// TIA Portal project "Plantilla_V18" (V18)

(* hardware
DEVICE "S71500/ET200MP station_1"  S7-1500 station
   slot 0: "Perfil soporte_0"  Rack  6ES7 590-1***0-0AA0
   slot 1: "PLC_1"  CPU 1516-3 PN/DP  6ES7 516-3AN01-0AB0  V2.1
      slot 3: "Display de la CPU_1"  6ES7591-1BA00-0AA0
   slot 2: "DI 32x24VDC HF_1"  DI 32x24VDC HF  6ES7 521-1BL00-0AB0  V2.1
   slot 3: "DQ 32x24VDC/0.5A HF_1"  DQ 32x24VDC/0.5A HF  6ES7 522-1BL01-0AB0  V1.0
   slot 4: "AI 8xU/I/RTD/TC ST_1"  AI 8xU/I/RTD/TC ST  6ES7 531-7KF00-0AB0  V2.1
   slot 5: "AQ 4xU/I ST_1"  AQ 4xU/I ST  6ES7 532-5HD00-0AB0  V2.1
*)

// ===== PLC "PLC_1"  CPU 1516-3 PN/DP =====

VAR_GLOBAL   // PLC tag table "Temporizadores y contadores"
   "Temp_barnizado" AT %T0 : Timer;
   "Temp_secado1_normal" AT %T1 : Timer;
   "Temp_pickandplace_s1" AT %T2 : Timer;
   "Temp_grabado_normal_p" AT %T4 : Timer;
   "Temp_grabado_lim_p" AT %T5 : Timer;
   "Temp_grabado_pickandplace" AT %T6 : Timer;
   "Temp_secado1_lim" AT %T7 : Timer;
   "Temp_secado1_pickandplace" AT %T8 : Timer;
   "Temp_plataforma_s1" AT %T9 : Timer;
   "Temp_plataforma_lectura_s1" AT %T10 : Timer;
   "Temp_pintado_lim" AT %T11 : Timer;
   "Temp_cinta" AT %T12 : Timer;
   "Contador_lecturas_defectuosas" AT %Z0 : Counter;
   "Temp_fugaz_21" AT %T13 : Timer;
   "Temp_plataforma_p" AT %T14 : Timer;
   "Temp_plataforma_b" AT %T15 : Timer;
   "Temp_plataforma_lectura_p" AT %T16 : Timer;
   "Temp_plataforma_lectura_b" AT %T17 : Timer;
   "Temp_pickandplace_p" AT %T18 : Timer;
   "Temp_pickandplace_b" AT %T19 : Timer;
   "Temp_grabado_lim_b" AT %T20 : Timer;
   "Temp_grabado_normal_b" AT %T21 : Timer;
   "Temp_grabado_normal_s1" AT %T22 : Timer;
   "Temp_grabado_lim_s1" AT %T23 : Timer;
END_VAR

VAR_GLOBAL   // PLC tag table "Entradas"
   "ON" AT %E0.0 : Bool;
   "EMER" AT %E0.2 : Bool;
   "rearme" AT %E0.3 : Bool;
   "START" AT %E0.4 : Bool;
   "Tablero_ajedrez" AT %E1.2 : Bool;
   "Pieza_cogida_robpp_s1" AT %E6.4 : Bool;
   "fin_secado1" AT %E3.6 : Bool;
   "fin_grabado_p" AT %E3.7 : Bool;
   "fin_grabado_b" AT %E4.0 : Bool;
   "fin_grabado_s1" AT %E4.1 : Bool;
   "fin_pintado" AT %E4.2 : Bool;
   "Home_robpp_s1" AT %E4.3 : Bool;
   "Home_robpp_gs1" AT %E4.4 : Bool;
   "Home_robpp_gp" AT %E4.5 : Bool;
   "Home_robpp_gb" AT %E4.6 : Bool;
   "Home_robpp_p" AT %E4.7 : Bool;
   "lectura_correcta_s1" AT %E5.0 : Bool;
   "lectura_incorrecta_s1" AT %E5.1 : Bool;
   "entra_s1" AT %E5.2 : Bool;
   "sigue_s1" AT %E5.3 : Bool;
   "vel_cinta_muestreada_bits" AT %EW4 : Int;
   "lectura_correcta_p" AT %E5.4 : Bool;
   "lectura_incorrecta_p" AT %E6.1 : Bool;
   "lectura_correcta_b" AT %E6.2 : Bool;
   "lectura_incorrecta_b" AT %E6.3 : Bool;
   "entra_p" AT %E6.5 : Bool;
   "sigue_p" AT %E6.7 : Bool;
   "entra_b" AT %E7.0 : Bool;
   "sigue_b" AT %E7.1 : Bool;
   "Pieza_cogida_robpp_gp" AT %E7.2 : Bool;
   "Pieza_cogida_robpp_gb" AT %E7.3 : Bool;
END_VAR

VAR_GLOBAL   // PLC tag table "Salidas"
   "Barnizar" AT %A0.0 : Bool;
   "Pintar" AT %A0.1 : Bool;
   "Secar" AT %A0.2 : Bool;
   "Robot_coger" AT %A0.3 : Bool;
   "Robot_dejar" AT %A0.4 : Bool;
   "Robot_reposo" AT %A0.5 : Bool;
   "Grabar" AT %A0.6 : Bool;
   "aviso_error_barnizado" AT %A0.7 : Bool;
   "aviso_fin_barnizado" AT %A1.1 : Bool;
   "aviso_error_secado1" AT %A1.2 : Bool;
   "aviso_fin_secado1" AT %A1.3 : Bool;
   "aviso_fin_pintado" AT %A1.4 : Bool;
   "aviso_error_grabado_p" AT %A1.5 : Bool;
   "aviso_fin_grabado_p" AT %A1.6 : Bool;
   "Robot_izq" AT %A1.7 : Bool;
   "Robot_delante" AT %A2.0 : Bool;
   "Robot_dcha" AT %A2.1 : Bool;
   "aviso_fin_pickandplace" AT %A2.2 : Bool;
   "aviso_errorT_pickandplace" AT %A2.3 : Bool;
   "aviso_errorConf_pickandplace" AT %A2.4 : Bool;
   "aviso_al_pp_coger_pieza_grabado_p" AT %A2.5 : Bool;
   "aviso_al_pp_coger_pieza_secado1" AT %A2.6 : Bool;
   "Leer" AT %A2.7 : Bool;
   "giro_ruedas_por_defecto" AT %A3.0 : Bool;
   "giro_ruedas_izquierda" AT %A3.1 : Bool;
   "aviso_errorT_lectura_plataforma_s1" AT %A3.2 : Bool;
   "avisor_errorT_plataforma_s1" AT %A3.3 : Bool;
   "aviso_fin_entrada_s1" AT %A3.4 : Bool;
   "aviso_fin_noEntra_s1" AT %A3.5 : Bool;
   "aviso_error_lectura_plataforma" AT %A3.6 : Bool;
   "aviso_error_pintado" AT %A1.0 : Bool;
   "cinta_sentido_antihorario" AT %A3.7 : Bool;
   "aviso_error_cinta" AT %A4.0 : Bool;
   "aviso_fin_cinta" AT %A4.1 : Bool;
   "Luz_Roja" AT %A4.2 : Bool;
   "aviso_fin_entrada_p" AT %A4.3 : Bool;
   "aviso_fin_entrada_b" AT %A4.4 : Bool;
   "aviso_fin_noEntra_p" AT %A4.5 : Bool;
   "aviso_fin_noEntra_b" AT %A4.6 : Bool;
   "aviso_fin_grabado_b" AT %A4.7 : Bool;
   "aviso_error_grabado_b" AT %A5.0 : Bool;
   "aviso_al_pp_coger_pieza_grabado_b" AT %A5.1 : Bool;
   "aviso_fin_grabado_s1" AT %A5.2 : Bool;
   "aviso_error_grabado_s1" AT %A5.3 : Bool;
   "aviso_al_pp_coger_pieza_grabsecado1" AT %A5.4 : Bool;
END_VAR

VAR_GLOBAL   // PLC tag table "Memorias"
   "M_flanco" AT %M0.0 : Bool;
   "PON" AT %M0.1 : Bool;
   "X0" AT %M0.2 : Bool;
   "X_ON" AT %M0.3 : Bool;
   "X_OFF" AT %M0.4 : Bool;
   "XM1" AT %M0.5 : Bool;
   "X1" AT %M0.6 : Bool;
   "XM2" AT %M0.7 : Bool;
   "X2" AT %M1.0 : Bool;
   "XM3" AT %M1.1 : Bool;
   "X3" AT %M1.2 : Bool;
   "XM4.1" AT %M1.3 : Bool;
   "X4.1" AT %M1.4 : Bool;
   "XM5.1" AT %M1.5 : Bool;
   "X5.1" AT %M1.6 : Bool;
   "XM6.1" AT %M1.7 : Bool;
   "X6.1" AT %M2.0 : Bool;
   "OFF" AT %E0.1 : Bool;
   "X_EMER" AT %M2.1 : Bool;
   "X10" AT %M2.2 : Bool;
   "X_PintadoModoCuadricula" AT %M2.3 : Bool;
   "X_PintadoModoNormal" AT %M2.4 : Bool;
   "X20" AT %M2.5 : Bool;
   "X21" AT %M2.6 : Bool;
   "X22" AT %M2.7 : Bool;
   "lectura_defectuosa" AT %M3.0 : Bool;
   "evento_lecturas" AT %M3.1 : Bool;
   "X23" AT %M3.2 : Bool;
   "XM7" AT %M3.3 : Bool;
   "X7" AT %M3.4 : Bool;
   "XM4.2" AT %M3.5 : Bool;
   "X4.2" AT %M3.6 : Bool;
   "XM4.3" AT %M3.7 : Bool;
   "X4.3" AT %M4.0 : Bool;
   "XM5.2" AT %M4.1 : Bool;
   "X5.2" AT %M4.2 : Bool;
   "XM5.3" AT %M4.3 : Bool;
   "X5.3" AT %M4.4 : Bool;
   "XM5.4" AT %M4.5 : Bool;
   "X5.4" AT %M4.6 : Bool;
   "X6.2" AT %M4.7 : Bool;
   "XM6.2" AT %M5.0 : Bool;
   "X6.3" AT %M5.1 : Bool;
   "XM6.3" AT %M5.2 : Bool;
   "X5.5" AT %M5.3 : Bool;
   "X5.6" AT %M5.4 : Bool;
   "X5.7" AT %M5.5 : Bool;
   "X5.8" AT %M5.6 : Bool;
   "XM5.5" AT %M5.7 : Bool;
   "XM5.6" AT %M6.0 : Bool;
   "XM5.7" AT %M6.1 : Bool;
   "XM5.8" AT %M6.2 : Bool;
END_VAR

VAR_GLOBAL   // PLC tag table "Entradas_SP"
   "SP_pintado_LaminaEnMesa" AT %E0.5 : Bool;
   "SP_barnizado_in" AT %E0.6 : Bool;
   "SP_secado1" AT %E0.7 : Bool;
   "SP_barnizado_out" AT %E1.3 : Bool;
   "SP_lectura_p" AT %E2.1 : Bool;
   "SP_lectura_b" AT %E2.2 : Bool;
   "SP_lectura_s1" AT %E2.3 : Bool;
   "SP_pickandplace_p_in" AT %E2.4 : Bool;
   "SP_pickandplace_p_out" AT %E2.5 : Bool;
   "SP_pickandplace_gp_in" AT %E2.6 : Bool;
   "SP_pickandplace_gp_out" AT %E2.7 : Bool;
   "SP_grabado_p" AT %E3.0 : Bool;
   "SP_grabado_b" AT %E3.1 : Bool;
   "SP_pickandplace_s1_in" AT %E6.0 : Bool;
   "SP_pickandplace_s1_out" AT %E1.1 : Bool;
   "SP_pickandplace_gs1_in" AT %E1.5 : Bool;
   "SP_pickandplace_gs1_out" AT %E3.2 : Bool;
   "SP_grabado_s1" AT %E3.3 : Bool;
   "SP_pickandplace_gb_in" AT %E3.4 : Bool;
   "SP_pickandplace_gb_out" AT %E3.5 : Bool;
   "SP_pintado_PiezaEnMesa" AT %E1.4 : Bool;
   "SP_pintado_LaminaEnOrigen" AT %E6.6 : Bool;
END_VAR

DATA_BLOCK "Datos_produccion"   // DB1
{ S7_Optimized_Access := 'TRUE' }
VERSION : 0.1
   VAR
      t_lim_respuesta_lectura : S5Time := S5T#10s;
      t_lim_plat_omni : S5Time := S5T#60s;
      t_lim_barnizado : S5Time := S5T#10s;
      t_lim_secado : S5Time := S5T#60s;
      t_normal_secado : S5Time := S5T#10s;
      t_lim_pickandplace : S5Time := S5T#60s;
      t_lim_robotpintado : S5Time := S5T#10s;
      t_lim_grabado : S5Time := S5T#60s;
      t_normal_grabado : S5Time := S5T#15s;
      t_lim_cinta : S5Time := S5T#10s;
      max_malas_lecturas : Word := 30;
      t_fugaz_21 : S5Time := S5T#1s;
      t_lim_pintado : S5Time;
   END_VAR
BEGIN
END_DATA_BLOCK

DATA_BLOCK "Datos_ModoCuadricula"   // DB20
{ S7_Optimized_Access := 'TRUE' }
VERSION : 0.1
   VAR
      t_lim_pintado_ModoCuadricula : S5Time := S5T#600s;
   END_VAR
BEGIN
END_DATA_BLOCK

DATA_BLOCK "Datos_ModoNormal"   // DB21
{ S7_Optimized_Access := 'TRUE' }
VERSION : 0.1
   VAR
      t_lim_pintado_ModoNormal : S5Time := S5T#180s;
   END_VAR
BEGIN
END_DATA_BLOCK

// folder: Barnizado

DATA_BLOCK "maniobra_barnizado_DB"   // DB2
{ S7_Optimized_Access := 'TRUE' }
VERSION : 0.1
// stored: InstanceOfName maniobra_barnizado
"maniobra_barnizado"
BEGIN
END_DATA_BLOCK

// folder: Cinta

DATA_BLOCK "maniobra_cinta_DB"   // DB8
{ S7_Optimized_Access := 'TRUE' }
VERSION : 0.1
// stored: InstanceOfName maniobra_cinta
"maniobra_cinta"
BEGIN
END_DATA_BLOCK

// folder: Entrada_a_estacion

DATA_BLOCK "maniobra_plataforma_omnidireccional_DB"   // DB6
{ S7_Optimized_Access := 'TRUE' }
VERSION : 0.1
// stored: InstanceOfName maniobra_plataforma_omnidireccional
"maniobra_plataforma_omnidireccional"
BEGIN
END_DATA_BLOCK

DATA_BLOCK "man_plat_omni_DB_Entrada_Pintado"   // DB7
{ S7_Optimized_Access := 'TRUE' }
VERSION : 0.1
// stored: InstanceOfName maniobra_plataforma_omnidireccional
"maniobra_plataforma_omnidireccional"
BEGIN
END_DATA_BLOCK

DATA_BLOCK "man_plat_omni_DB_Entrada_Barnizado"   // DB10
{ S7_Optimized_Access := 'TRUE' }
VERSION : 0.1
// stored: InstanceOfName maniobra_plataforma_omnidireccional
"maniobra_plataforma_omnidireccional"
BEGIN
END_DATA_BLOCK

// folder: Grabado_y_secado

DATA_BLOCK "maniobra_secado_DB"   // DB4
{ S7_Optimized_Access := 'TRUE' }
VERSION : 0.1
// stored: InstanceOfName maniobra_grabado_secado
"maniobra_grabado_secado"
BEGIN
END_DATA_BLOCK

DATA_BLOCK "maniobra_grabado_DB"   // DB5
{ S7_Optimized_Access := 'TRUE' }
VERSION : 0.1
// stored: InstanceOfName maniobra_grabado_secado
"maniobra_grabado_secado"
BEGIN
END_DATA_BLOCK

DATA_BLOCK "man_grabado_b"   // DB14
{ S7_Optimized_Access := 'TRUE' }
VERSION : 0.1
// stored: InstanceOfName maniobra_grabado_secado
"maniobra_grabado_secado"
BEGIN
END_DATA_BLOCK

// folder: Pick_and_place

DATA_BLOCK "maniobra_pickandplace_DB"   // DB3
{ S7_Optimized_Access := 'TRUE' }
VERSION : 0.1
// stored: InstanceOfName maniobra_pickandplace
"maniobra_pickandplace"
BEGIN
END_DATA_BLOCK

DATA_BLOCK "man_pickandplace_gp1"   // DB11
{ S7_Optimized_Access := 'TRUE' }
VERSION : 0.1
// stored: InstanceOfName maniobra_pickandplace
"maniobra_pickandplace"
BEGIN
END_DATA_BLOCK

DATA_BLOCK "man_pickandplace_gp2"   // DB12
{ S7_Optimized_Access := 'TRUE' }
VERSION : 0.1
// stored: InstanceOfName maniobra_pickandplace
"maniobra_pickandplace"
BEGIN
END_DATA_BLOCK

DATA_BLOCK "man_pickandplace_gb1"   // DB13
{ S7_Optimized_Access := 'TRUE' }
VERSION : 0.1
// stored: InstanceOfName maniobra_pickandplace
"maniobra_pickandplace"
BEGIN
END_DATA_BLOCK

DATA_BLOCK "man_pickandplace_gb2"   // DB15
{ S7_Optimized_Access := 'TRUE' }
VERSION : 0.1
// stored: InstanceOfName maniobra_pickandplace
"maniobra_pickandplace"
BEGIN
END_DATA_BLOCK

DATA_BLOCK "man_pickandplace_s1_2"   // DB16
{ S7_Optimized_Access := 'TRUE' }
VERSION : 0.1
// stored: InstanceOfName maniobra_pickandplace
"maniobra_pickandplace"
BEGIN
END_DATA_BLOCK

DATA_BLOCK "man_pickandplace_gs1_1"   // DB17
{ S7_Optimized_Access := 'TRUE' }
VERSION : 0.1
// stored: InstanceOfName maniobra_pickandplace
"maniobra_pickandplace"
BEGIN
END_DATA_BLOCK

DATA_BLOCK "man_grabado_s1"   // DB18
{ S7_Optimized_Access := 'TRUE' }
VERSION : 0.1
// stored: InstanceOfName maniobra_grabado_secado
"maniobra_grabado_secado"
BEGIN
END_DATA_BLOCK

DATA_BLOCK "man_pickandplace_gs1_2"   // DB19
{ S7_Optimized_Access := 'TRUE' }
VERSION : 0.1
// stored: InstanceOfName maniobra_pickandplace
"maniobra_pickandplace"
BEGIN
END_DATA_BLOCK

// folder: Pintado

DATA_BLOCK "maniobra_pintado_DB_1"   // DB9
{ S7_Optimized_Access := 'TRUE' }
VERSION : 0.1
// stored: InstanceOfName maniobra_pintado
"maniobra_pintado"
BEGIN
END_DATA_BLOCK

// folder: (top level)

ORGANIZATION_BLOCK "Main"   // OB1, STL, ProgramCycle
TITLE = "Main Program Sweep (Cycle)"
{ S7_Optimized_Access := 'TRUE' }
VERSION : 0.1
   VAR_INPUT
      Initial_Call : Bool;   // Initial call of this OB
      Remanence : Bool;   // =True, if remanent data are available
   END_VAR
BEGIN

REGION Network 1: Llamada a los tests unitarios (comentado)
   //CALL  "test_barnizado"

   // CALL  "test_secado"
   //   CALL  "test_grabado"
   //     CALL  "test_pickandplace"
   //     CALL  "test_plataforma_omnidireccional"
   //      CALL  "test_cinta"
   //      CALL  "test_pintado"
   //      CALL  "Modos_pintado"

   //   CALL  "Emergencia"
END_REGION

REGION Network 2: Llamada a las FC
         CALL  "contador_fallos_lectura"
         ( max_malas_lecturas  := "Datos_produccion".max_malas_lecturas,
           debe_retirar_piezas := "evento_lecturas"
         );
         CALL  "gestion_fallos_lectura";
         CALL  "Emergencia";
         CALL  "Flancos";
         CALL  "Modos_pintado";
END_REGION

REGION Network 3: X0 -> XM
         A     "X0";
         A     "PON";
         AN    "OFF";
         S     "XM1";
         S     "XM2";
         S     "XM3";
         S     "XM4.1";
         S     "XM4.2";
         S     "XM4.3";
         S     "XM5.1";
         S     "XM6.1";
         S     "XM7";
         S     "X_ON";
         R     "X0";
END_REGION

REGION Network 4: X_ON -> X_OFF
         A     "X_ON";
         A     "OFF";
         S     "X_OFF";
         R     "X_ON";
END_REGION

REGION Network 5: X1, X2, X3, X4, X5, X6, X7, X_OFF -> X0
         A     "X1";
         A     "X2";
         A     "X3";
         A     "X4.1";
         S     "XM4.2";
         S     "XM4.3";
         A     "X5.1";
         A     "X6.1";
         A     "X7";
         A     "X_OFF";
         S     "X0";
         R     "X1";
         R     "X2";
         R     "X3";
         R     "X4.1";
         R     "X4.2";
         R     "X4.3";
         R     "X5.1";
         R     "X6.1";
         R     "X7";
         R     "X_OFF";
END_REGION

REGION Network 6: X1 -> XM1
         A     "X1";
         A     "SP_pintado_PiezaEnMesa";
         S     "XM1";
         R     "X1";
END_REGION

REGION Network 7: X2 -> XM2
         A     "X2";
         A     "SP_barnizado_in";
         S     "XM2";
         R     "X2";
END_REGION

REGION Network 8: X3 -> XM3
         A     "X3";
         A     "SP_secado1";
         S     "XM3";
         R     "XM3";
END_REGION

REGION Network 9: X4.1-> XM4.1
         A     "X4.1";
         A     "SP_grabado_p";
         S     "XM4.1";
         R     "X4.1";
END_REGION

REGION Network 10: X4.2 -> XM4.2
         A     "X4.2";
         A     "SP_grabado_b";
         S     "XM4.2";
         R     "X4.2";
END_REGION

REGION Network 11: X4.3 -> XM4.3
         A     "X4.3";
         A     "SP_grabado_s1";
         S     "XM4.3";
         R     "X4.3";
END_REGION

REGION Network 12: X5.1-> XM5.1
         A     "X5.1";
         A     "SP_pickandplace_gb_in";
         S     "XM5.1";
         R     "X5.1";
END_REGION

REGION Network 13: X5.2->XM5.2
         A     "X5.2";
         A     "SP_pickandplace_gp_in";
         S     "XM5.2";
         R     "X5.2";
END_REGION

REGION Network 14: X5.3->XM5.3
         A     "X5.3";
         A     "SP_pickandplace_gb_in";
         R     "X5.3";
         S     "XM5.3";
END_REGION

REGION Network 15: X5.4->XM5.4
         A     "X5.4";
         A     "aviso_al_pp_coger_pieza_grabado_b";
         S     "XM5.4";
         R     "X5.4";
END_REGION

REGION Network 16: X5.5->XM5.5
         A     "X5.5";
         A     "SP_pickandplace_s1_in";
         R     "X5.5";
         S     "XM5.5";
END_REGION

REGION Network 17: X5.6->XM5.6
         A     "X5.6";
         A     "aviso_al_pp_coger_pieza_secado1";
         R     "X5.6";
         S     "XM5.6";
END_REGION

REGION Network 18: X5.7->XM5.7
         A     "X5.7";
         A     "SP_pickandplace_gs1_in";
         R     "X5.7";
         S     "XM5.7";
END_REGION

REGION Network 19: X5.8->XM5.8
         A     "X5.8";
         A     "aviso_al_pp_coger_pieza_grabsecado1";
         R     "X5.8";
         S     "XM5.8";
END_REGION

REGION Network 20: X6.1 -> XM6.1
         A     "X6.1";
         A     "X_ON";
         S     "XM6.1";
         R     "X6.1";
END_REGION

REGION Network 21: X6.2 -> XM6.2
         A     "X6.2";
         A     "X_ON";
         R     "X6.2";
         S     "XM6.2";
END_REGION

REGION Network 22: X6.3 -> XM6.3
         A     "X6.3";
         A     "X_ON";
         R     "X6.3";
         S     "XM6.3";
END_REGION

REGION Network 23: X7 -> XM7
         A     "X7";
         A     "X_ON";
         R     "X7";
         S     "XM7";
END_REGION

REGION Network 24: XM1 -> X1 y tratamiento M1 (pintado)
         A     "XM1";
         JCN   _pintado;
         CALL  "maniobra_pintado", "maniobra_pintado_DB_1"
         ( SP_pieza              := "SP_pintado_PiezaEnMesa",
           SP_lamina_mesa        := "SP_pintado_LaminaEnMesa",
           SP_lamina_pos_inicial := "SP_pintado_LaminaEnOrigen",
           ModoLamina            := "X_PintadoModoCuadricula",
           ModoNormal            := "X_PintadoModoNormal",
           pintado_terminado     := "fin_pintado",
           RESET                 := false,
           t_lim_pintado_con_lam := "Datos_produccion".t_lim_pintado_ModoCuadricula,
           t_lim_pintado_sin_lam := "Datos_produccion".t_lim_pintado_ModoNormal,
           Temporizador_limite   := "Temp_pintado_lim",
           Tempor_pickandplace1  := "Temp_pickandplace_s1",
           Tempor_pickandplace2  := "Temp_pickandplace_s1",
           SP_pickandplace_in    := "SP_pickandplace_p_in",
           SP_pickandplace_out   := "SP_pickandplace_p_out",
           Sensor_home           := "Home_robpp_p",
           Lamina_cogida         := "Pieza_cogida_robpp_s1",
           t_lim_pickandplace    := "Datos_produccion".t_lim_pickandplace,
           Act_pintar            := "Pintar",
           bde_tiempo            := "aviso_error_pintado",
           bdf_correcta          := "aviso_fin_pintado"
         );

         A     "aviso_fin_pintado";
         S     "X1";
         R     "XM1";
   _pintado:NOP   0;
END_REGION

REGION Network 25: XM2 -> X2 y tratamiento M2 (barnizado)
         A     "XM2";
         JCN   _barnizado;
         CALL  "maniobra_barnizado", "maniobra_barnizado_DB"
         ( SP               := "SP_barnizado_in",
           indicador_de_fin := "SP_barnizado_out",
           t_lim            := "Datos_produccion".t_lim_barnizado,
           Temporizador     := "Temp_barnizado",
           RESET            := false,
           Actuador         := "Barnizar",
           bde_tiempo       := "aviso_error_barnizado",
           bdf_correcta     := "aviso_fin_barnizado"
         );

         A     "aviso_fin_barnizado";
         S     "X2";
         R     "XM2";

   _barnizado:NOP   0;
END_REGION

REGION Network 26: XM3 -> X3 y tratamiento M3 (secado)
         A     "XM3";
         JCN   _secado;
         CALL  "maniobra_grabado_secado", "maniobra_secado_DB"
         ( SP_maq                   := "SP_secado1",
           t_normal_maq             := "Datos_produccion".t_normal_secado,
           t_lim_man                := "Datos_produccion".t_lim_secado,
           RESET                    := false,
           Temp_normal_maq          := "Temp_secado1_normal",
           Temp_lim_maq             := "Temp_secado1_lim",
           bdf_correcta             := "aviso_fin_secado1",
           bde_Tiempo               := "aviso_error_secado1",
           aviso_a_robot_para_coger := "aviso_al_pp_coger_pieza_secado1",
           Actuador                 := "Secar"
         );
         A     "aviso_fin_secado1";
         S     "X3";
         R     "XM3";
   _secado:NOP   0;
END_REGION

REGION Network 27: XM4.1 -> X4.1 y tratamiento M4.1 (grabado del pintado)
         A     "XM4.1";
         JCN   _grabadopintado;
         CALL  "maniobra_grabado_secado", "maniobra_grabado_DB"
         ( SP_maq                   := "SP_grabado_p",
           t_normal_maq             := "Datos_produccion".t_normal_grabado,
           t_lim_man                := "Datos_produccion".t_lim_grabado,
           RESET                    := FALSE,
           Temp_normal_maq          := "Temp_grabado_normal_p",
           Temp_lim_maq             := "Temp_grabado_lim_p",
           bdf_correcta             := "aviso_fin_grabado_p",
           bde_Tiempo               := "aviso_error_grabado_p",
           aviso_a_robot_para_coger := "aviso_al_pp_coger_pieza_grabado_p",
           Actuador                 := "Grabar"
         );
         A     "aviso_fin_grabado_p";
         S     "X4.1";
         R     "XM4.1";
   _grabadopintado:NOP   0;
END_REGION

REGION Network 28: XM4.2 -> X4.2 y tratamiento M4.2 (grabado del barnizado)
         A     "XM4.2";
         JCN   _grabadobarnizado;
         CALL  "maniobra_grabado_secado", "man_grabado_b"
         ( SP_maq                   := "SP_grabado_b",
           t_normal_maq             := "Datos_produccion".t_normal_grabado,
           t_lim_man                := "Datos_produccion".t_lim_grabado,
           RESET                    := false,
           Temp_normal_maq          := "Temp_grabado_normal_b",
           Temp_lim_maq             := "Temp_grabado_lim_b",
           bdf_correcta             := "aviso_fin_grabado_b",
           bde_Tiempo               := "aviso_error_grabado_b",
           aviso_a_robot_para_coger := "aviso_al_pp_coger_pieza_grabado_b",
           Actuador                 := "Grabar"
         );
         A     "aviso_fin_grabado_b";
         S     "X4.2";
         R     "XM4.2";
   _grabadobarnizado:NOP   0;
END_REGION

REGION Network 29: XM4.3 -> X4.3 y tratamiento M4.3 (grabado del secado)
         A     "XM4.3";
         JCN   _grabadosecado;
         CALL  "maniobra_grabado_secado", "man_grabado_s1"
         ( SP_maq                   := "SP_grabado_s1",
           t_normal_maq             := "Datos_produccion".t_normal_grabado,
           t_lim_man                := "Datos_produccion".t_lim_grabado,
           RESET                    := false,
           Temp_normal_maq          := "Temp_grabado_normal_s1",
           Temp_lim_maq             := "Temp_grabado_lim_s1",
           bdf_correcta             := "aviso_fin_grabado_s1",
           bde_Tiempo               := "aviso_error_grabado_s1",
           aviso_a_robot_para_coger := "aviso_al_pp_coger_pieza_grabsecado1",
           Actuador                 := "Grabar"
         );
         A     "aviso_fin_grabado_s1";
         S     "X4.3";
         R     "XM4.3";
   _grabadosecado:NOP   0;
END_REGION

REGION Network 30: XM5.1->X5.1 y tratamiento M5.1 (pick and place para dejar pieza en la grabadora pintado)
         A     "XM5.1";
         JCN   _pickandplace_grabadopintado1;
         CALL  "maniobra_pickandplace", "man_pickandplace_gp1"
         ( SP1          := "SP_pickandplace_gb_in",
           P_cogida     := "Pieza_cogida_robpp_gp",
           S_home       := "Home_robpp_gp",
           t_lim        := "Datos_produccion".t_lim_pickandplace,
           Temporizador := "Temp_pickandplace_p",
           RESET        := false,
           SP2          := "SP_grabado_p",
           Mov1         := "Robot_coger",
           Mov2         := "Robot_delante",
           Mov4         := "Robot_reposo",
           bdf_correcta := "aviso_fin_pickandplace",
           bde_tiempo   := "aviso_errorT_pickandplace",
           bde_config   := "aviso_errorConf_pickandplace",
           Mov0         := "Robot_izq",
           Mov3         := "Robot_dejar"
         );
         A     "aviso_fin_pickandplace";
         S     "X5.1";
         R     "XM5.1";
   _pickandplace_grabadopintado1:NOP   0;
END_REGION

REGION Network 31: XM5.2->X5.2 y tratamiento M5.2 (pick and place para recoger la pieza de la grabadora de pintado)
         A     "XM5.2";
         JCN   _pickandplace_grabadopintado2;
         CALL  "maniobra_pickandplace", "man_pickandplace_gp1"
         ( SP1          := "SP_pickandplace_gp_in",
           P_cogida     := "Pieza_cogida_robpp_gp",
           S_home       := "Home_robpp_gp",
           t_lim        := "Datos_produccion".t_lim_pickandplace,
           Temporizador := "Temp_pickandplace_p",
           RESET        := false,
           SP2          := "SP_grabado_p",
           Mov1         := "Robot_coger",
           Mov2         := "Robot_delante",
           Mov4         := "Robot_reposo",
           bdf_correcta := "aviso_fin_pickandplace",
           bde_tiempo   := "aviso_errorT_pickandplace",
           bde_config   := "aviso_errorConf_pickandplace",
           Mov0         := "Robot_izq",
           Mov3         := "Robot_dejar"
         );
         A     "aviso_fin_pickandplace";
         R     "XM5.2";
         S     "X5.2";
   _pickandplace_grabadopintado2:NOP   0;
END_REGION

REGION Network 32: XM5.3->X5.3 y tratamiento M5.3 (pick and place para meter la pieza en la grabadora de barnizado)
         A     "XM5.3";
         JCN   _pickandplace_grabado_barnizado1;
         CALL  "maniobra_pickandplace", "man_pickandplace_gb1"
         ( SP1          := "SP_pickandplace_gb_in",
           P_cogida     := "Pieza_cogida_robpp_gb",
           S_home       := "Home_robpp_gb",
           t_lim        := "Datos_produccion".t_lim_pickandplace,
           Temporizador := "Temp_pickandplace_b",
           RESET        := false,
           SP2          := "SP_grabado_b",
           Mov1         := "Robot_coger",
           Mov2         := "Robot_delante",
           Mov4         := "Robot_reposo",
           bdf_correcta := "aviso_fin_pickandplace",
           bde_tiempo   := "aviso_errorT_pickandplace",
           bde_config   := "aviso_errorConf_pickandplace",
           Mov0         := "Robot_izq",
           Mov3         := "Robot_dejar"
         );
         A     "aviso_fin_pickandplace";
         S     "X5.3";
         R     "XM5.3";
   _pickandplace_grabado_barnizado1:NOP   0;
END_REGION

REGION Network 33: XM5.4->X5.4 y tratamiento M5.4 (pick and place para recoger la pieza del grabado del barnizado)
         A     "XM5.4";
         JCN   _pickandplace_grabado_barnizado2;
         CALL  "maniobra_pickandplace", "man_pickandplace_gb2"
         ( SP1          := "aviso_al_pp_coger_pieza_grabado_b",
           P_cogida     := "Pieza_cogida_robpp_gb",
           S_home       := "Home_robpp_gb",
           t_lim        := "Datos_produccion".t_lim_pickandplace,
           Temporizador := "Temp_pickandplace_b",
           RESET        := false,
           SP2          := "SP_pickandplace_gb_out",
           Mov1         := "Robot_coger",
           Mov2         := "Robot_dcha",
           Mov4         := "Robot_reposo",
           bdf_correcta := "aviso_fin_pickandplace",
           bde_tiempo   := "aviso_errorT_pickandplace",
           bde_config   := "aviso_errorConf_pickandplace",
           Mov0         := "Robot_delante",
           Mov3         := "Robot_dejar"
         );
         A     "aviso_fin_pickandplace";
         S     "X5.4";
         R     "XM5.4";
   _pickandplace_grabado_barnizado2:NOP   0;
END_REGION

REGION Network 34: XM5.5->X5.5 y tratamiento M5.5 (pick and place para meter la pieza en la máquina de secado)
         A     "XM5.5";
         JCN   _pickandplace_secado1;
         CALL  "maniobra_pickandplace", "maniobra_pickandplace_DB"
         ( SP1          := "SP_pickandplace_s1_in",
           P_cogida     := "Pieza_cogida_robpp_s1",
           S_home       := "Home_robpp_s1",
           t_lim        := "Datos_produccion".t_lim_pickandplace,
           Temporizador := "Temp_pickandplace_s1",
           RESET        := FALSE,
           SP2          := "SP_secado1",
           Mov1         := "Robot_coger",
           Mov2         := "Robot_delante",
           Mov4         := "Robot_reposo",
           bdf_correcta := "aviso_fin_pickandplace",
           bde_tiempo   := "aviso_errorT_pickandplace",
           bde_config   := "aviso_errorConf_pickandplace",
           Mov0         := "Robot_izq",
           Mov3         := "Robot_dejar"
         );
         A     "aviso_fin_pickandplace";
         R     "XM5.5";
         S     "X5.5";
   _pickandplace_secado1:NOP   0;
END_REGION

REGION Network 35: XM5.6->X5.6 y tratamiento M5.6 (pick and place para sacar la pieza de la máquina de secado)
         A     "XM5.6";
         JCN   _pickandplace_secado2;
         CALL  "maniobra_pickandplace", "man_pickandplace_s1_2"
         ( SP1          := "aviso_al_pp_coger_pieza_secado1",
           P_cogida     := "Pieza_cogida_robpp_s1",
           S_home       := "Home_robpp_s1",
           t_lim        := "Datos_produccion".t_lim_pickandplace,
           Temporizador := "Temp_pickandplace_s1",
           RESET        := false,
           SP2          := "SP_pickandplace_s1_out",
           Mov1         := "Robot_coger",
           Mov2         := "Robot_dcha",
           Mov4         := "Robot_reposo",
           bdf_correcta := "aviso_fin_pickandplace",
           bde_tiempo   := "aviso_errorT_pickandplace",
           bde_config   := "aviso_errorConf_pickandplace",
           Mov0         := "Robot_delante",
           Mov3         := "Robot_dejar"
         );
         A     "aviso_fin_pickandplace";
         R     "XM5.6";
         S     "X5.6";
   _pickandplace_secado2:NOP   0;
END_REGION

REGION Network 36: XM5.7->X5.7 y tratamiento M5.7 (pick and place para meter la pieza en la grabadora de secado)
         A     "XM5.7";
         JCN   _pickandplace_grabado_secado1;
         CALL  "maniobra_pickandplace", "man_pickandplace_gs1_1"
         ( SP1          := "SP_pickandplace_gs1_in",
           P_cogida     := "Pieza_cogida_robpp_s1",
           S_home       := "Home_robpp_s1",
           t_lim        := "Datos_produccion".t_lim_pickandplace,
           Temporizador := "Temp_pickandplace_s1",
           RESET        := false,
           SP2          := "SP_grabado_s1",
           Mov1         := "Robot_coger",
           Mov2         := "Robot_delante",
           Mov4         := "Robot_reposo",
           bdf_correcta := "aviso_fin_pickandplace",
           bde_tiempo   := "aviso_errorT_pickandplace",
           bde_config   := "aviso_errorConf_pickandplace",
           Mov0         := "Robot_izq",
           Mov3         := "Robot_dejar"
         );
         A     "aviso_fin_pickandplace";
         R     "XM5.7";
         S     "X5.7";
   _pickandplace_grabado_secado1:NOP   0;
END_REGION

REGION Network 37: XM5.78->X5.8 y tratamiento M5.8 (pick and place para sacar la pieza de la grabadora de secado)
         A     "XM5.8";
         JCN   _pickandplace_grabado_secado2;
         CALL  "maniobra_pickandplace", "man_pickandplace_gs1_2"
         ( SP1          := "aviso_al_pp_coger_pieza_grabsecado1",
           P_cogida     := "Pieza_cogida_robpp_s1",
           S_home       := "Home_robpp_s1",
           t_lim        := "Datos_produccion".t_lim_pickandplace,
           Temporizador := "Temp_pickandplace_s1",
           RESET        := false,
           SP2          := "SP_pickandplace_gs1_out",
           Mov1         := "Robot_coger",
           Mov2         := "Robot_dcha",
           Mov4         := "Robot_reposo",
           bdf_correcta := "aviso_fin_pickandplace",
           bde_tiempo   := "aviso_errorT_pickandplace",
           bde_config   := "aviso_errorConf_pickandplace",
           Mov0         := "Robot_delante",
           Mov3         := "Robot_dejar"
         );
         A     "aviso_fin_pickandplace";
         S     "X5.8";
         R     "XM5.8";

   _pickandplace_grabado_secado2:NOP   0;
END_REGION

REGION Network 38: XM6.1 -> X6.1 y tratamiento M6.1 (entrada a estación de pintado)
         A     "XM6.1";
         JCN   _entrada_pintado;
         CALL  "maniobra_plataforma_omnidireccional", "man_plat_omni_DB_Entrada_Pintado"
         ( SP                          := "SP_lectura_p",
           Lectura_correcta            := "lectura_correcta_p",
           Lectura_incorrecta          := "lectura_incorrecta_p",
           Entra_estacion              := "entra_p",
           Sigue_cinta                 := "sigue_p",
           SP_estacion                 := "SP_pickandplace_p_in",
           RESET                       := false,
           t_lim_lectura               := "Datos_produccion".t_lim_respuesta_lectura,
           t_lim_maniobra              := "Datos_produccion".t_lim_plat_omni,
           Temp_lectura                := "Temp_plataforma_lectura_p",
           Temp_maniobra               := "Temp_plataforma_p",
           Actuador_ruedas_por_defecto := "giro_ruedas_por_defecto",
           Actuador_lectura            := "Leer",
           Actuador_ruedas_giro        := "giro_ruedas_izquierda",
           bde_tiempo_lectura          := "aviso_errorT_lectura_plataforma_s1",
           bde_tiempo                  := "aviso_errorT_lectura_plataforma_s1",
           bde_lectura                 := "aviso_error_lectura_plataforma",
           bdf_piezadentro             := "aviso_fin_entrada_p",
           bdf_piezasiguerecto         := "aviso_fin_noEntra_p"
         );

         A     "aviso_fin_entrada_p";
         O     "aviso_fin_entrada_p";
         R     "XM6.1";
         S     "X6.1";
   _entrada_pintado:NOP   0;
END_REGION

REGION Network 39: XM6.2 -> X6.2 y tratamiento M6.2 (entrada a estación de barnizado)
         A     "XM6.2";
         JCN   _entrada_barnizado;
         CALL  "maniobra_plataforma_omnidireccional", "man_plat_omni_DB_Entrada_Barnizado"
         ( SP                          := "SP_lectura_b",
           Lectura_correcta            := "lectura_correcta_b",
           Lectura_incorrecta          := "lectura_incorrecta_b",
           Entra_estacion              := "entra_b",
           Sigue_cinta                 := "sigue_b",
           SP_estacion                 := "SP_barnizado_in",
           RESET                       := false,
           t_lim_lectura               := "Datos_produccion".t_lim_respuesta_lectura,
           t_lim_maniobra              := "Datos_produccion".t_lim_plat_omni,
           Temp_lectura                := "Temp_plataforma_lectura_b",
           Temp_maniobra               := "Temp_plataforma_b",
           Actuador_ruedas_por_defecto := "giro_ruedas_por_defecto",
           Actuador_lectura            := "Leer",
           Actuador_ruedas_giro        := "giro_ruedas_izquierda",
           bde_tiempo_lectura          := "aviso_errorT_lectura_plataforma_s1",
           bde_tiempo                  := "aviso_errorT_lectura_plataforma_s1",
           bde_lectura                 := "aviso_error_lectura_plataforma",
           bdf_piezadentro             := "aviso_fin_entrada_b",
           bdf_piezasiguerecto         := "aviso_fin_noEntra_b"
         );
         A     "aviso_fin_entrada_b";
         O     "aviso_fin_noEntra_b";
         R     "XM6.2";
         S     "X6.2";
   _entrada_barnizado:NOP   0;
END_REGION

REGION Network 40: XM6.3 -> X6.3 y tratamiento M6.3 (entrada a estación de secado)
         A     "XM6.3";
         JCN   _entrada_secado;
         CALL  "maniobra_plataforma_omnidireccional", "maniobra_plataforma_omnidireccional_DB"
         ( SP                          := "SP_lectura_s1",
           Lectura_correcta            := "lectura_correcta_s1",
           Lectura_incorrecta          := "lectura_incorrecta_s1",
           Entra_estacion              := "entra_s1",
           Sigue_cinta                 := "sigue_s1",
           SP_estacion                 := "SP_pickandplace_s1_in",
           RESET                       := false,
           t_lim_lectura               := "Datos_produccion".t_lim_respuesta_lectura,
           t_lim_maniobra              := "Datos_produccion".t_lim_plat_omni,
           Temp_lectura                := "Temp_plataforma_lectura_s1",
           Temp_maniobra               := "Temp_plataforma_s1",
           Actuador_ruedas_por_defecto := "giro_ruedas_por_defecto",
           Actuador_lectura            := "Leer",
           Actuador_ruedas_giro        := "giro_ruedas_izquierda",
           bde_tiempo_lectura          := "aviso_errorT_lectura_plataforma_s1",
           bde_tiempo                  := "avisor_errorT_plataforma_s1",
           bde_lectura                 := "aviso_error_lectura_plataforma",
           bdf_piezadentro             := "aviso_fin_entrada_s1",
           bdf_piezasiguerecto         := "aviso_fin_noEntra_s1"
         );
         A     "aviso_fin_entrada_s1";
         O     "aviso_fin_noEntra_s1";
         R     "XM6.3";
         S     "X6.3";
   _entrada_secado:NOP   0;
END_REGION

REGION Network 41: XM7 -> X7 y tratamiento de M7 (cinta)
         A     "XM7";
         JCN   _cinta;
         CALL  "maniobra_cinta", "maniobra_cinta_DB"
         ( vel_cinta_bits      := "vel_cinta_muestreada_bits",
           t_lim               := "Datos_produccion".t_lim_cinta,
           Temporizador        := "Temp_cinta",
           RESET               := "EMER",
           Sentido_antihorario := "cinta_sentido_antihorario",
           bdf_correcta        := "aviso_fin_cinta",
           bde_velocidad       := "aviso_error_cinta"
         );
         A     "aviso_fin_cinta";
         R     "XM7";
         S     "X7";
   _cinta:NOP   0;
END_REGION
END_ORGANIZATION_BLOCK

ORGANIZATION_BLOCK "Startup"   // OB100, STL, Startup
TITLE = "Complete Restart"
{ S7_Optimized_Access := 'TRUE' }
VERSION : 0.1
   VAR_INPUT
      LostRetentive : Bool;   // True if retentive data are lost
      LostRTC : Bool;   // True if date and time are lost
   END_VAR
BEGIN

REGION Network 1
         SET;
         S     "X0";
         S     "X10";
         S     "X20";
         R     "X_PintadoModoCuadricula";
         R     "X_PintadoModoNormal";
         R     "X_EMER";
         R     "X21";
         R     "X22";
END_REGION
END_ORGANIZATION_BLOCK

// folder: Barnizado

FUNCTION_BLOCK "maniobra_barnizado"   // FB2, STL
{ S7_Optimized_Access := 'TRUE' }
VERSION : 0.1
// Para reciclar código, se utiliza una misma maniobra para las máquinas de barnizado, grabado y secado.
   VAR_INPUT
      SP : Bool;
      indicador_de_fin : Bool;
      t_lim : S5Time := S5T#0ms;
      Temporizador : Timer;
      RESET : Bool;
   END_VAR
   VAR_OUTPUT
      Actuador : Bool;
      bde_tiempo : Bool;
      bdf_correcta : Bool;
   END_VAR
   VAR
      bdt : Bool;
      XE2 : Bool;
      X1 : Bool;
      XS2 : Bool;
      X_Err_Tiempo : Bool;
   END_VAR
BEGIN

REGION Network 1: Desconexión por RESET
         A     #RESET;
   //resetar los bits
         R     #bdt;
         R     #bde_tiempo;
         R     #bdf_correcta;
   //resetar temporizador
         R     #Temporizador;
         FR    #Temporizador;
   //resetar actuadores
         R     #Actuador;
         BEC;
END_REGION

REGION Network 2: Desconexión por error síncrono (exceso de tiempo)
         A     #X_Err_Tiempo;
         S     #bde_tiempo;
   //R     #X_Err_Tiempo
         R     #bdt;
         R     #bdf_correcta;
         R     #Temporizador;
         FR    #Temporizador;
         R     #Actuador;
         BEC;
END_REGION

REGION Network 3: Desconexión por finalización correcta
         A     #XS2;
         S     #bdf_correcta;
         R     #XS2;
         R     #bdt;
         R     #bde_tiempo;
         R     #Temporizador;
         FR    #Temporizador;
         R     #Actuador;
         BEC;
END_REGION

REGION Network 4: Conexión/ arranque de la maniobra
         SET;
         FP    #bdt;
         R     #bde_tiempo;
   //  R     #bdf_correcta
         S     #XE2;
         R     #X1;
         R     #XS2;
         R     #X_Err_Tiempo;
END_REGION

REGION Network 5: E2 -> X1
         A     #XE2;
         A     #SP;
         S     #X1;
         R     #XE2;
END_REGION

REGION Network 6: Definir perro guardián
         A     #X1;
         L     #t_lim;
         SS    #Temporizador;
END_REGION

REGION Network 7: X1-> XS2
         A     #X1;
         A     #indicador_de_fin;
         S     #XS2;
         R     #X1;
END_REGION

REGION Network 8: Activación del perro guardián
         A     #Temporizador;
         =     #X_Err_Tiempo;
END_REGION

REGION Network 9: Tratamiento X1
         A     #X1;
         =     #Actuador;
END_REGION
END_FUNCTION_BLOCK

// folder: Cinta

FUNCTION_BLOCK "maniobra_cinta"   // FB5, STL
{ S7_Optimized_Access := 'TRUE' }
VERSION : 0.1
   VAR_INPUT
      vel_cinta_bits : Int;
      t_lim : S5Time;
      Temporizador : Timer;
      RESET : Bool;
   END_VAR
   VAR_OUTPUT
      Sentido_antihorario : Bool;
      bdf_correcta : Bool;
      bde_velocidad : Bool;
   END_VAR
   VAR
      E7 : Bool;
      X1 : Bool;
      X2 : Bool;
      X_Err_Cinta : Bool;
      S7 : Bool;
      bdt : Bool;
      fuera_rango : Bool;
   END_VAR
   VAR_TEMP
      ret_val_scale : Word;
      vel_cinta_rpm : Real;
   END_VAR
BEGIN

REGION Network 1: Desconexión por RESET
         A     #RESET;
         R     #bdt;
         R     #bde_velocidad;
         R     #bdf_correcta;
         R     #Temporizador;
         FR    #Temporizador;
         R     #Sentido_antihorario;
         R     #fuera_rango;
         BEC;
END_REGION

REGION Network 2: Desconexión por velocidad de la cinta fuera de los rangos de lectura permitidos por el sensor
         A     #X_Err_Cinta;
         S     #bde_velocidad;
   // R     #X_Err_Cinta
         R     #bdt;
         R     #bdf_correcta;
         R     #Temporizador;
         FR    #Temporizador;
         R     #Sentido_antihorario;
         R     #fuera_rango;
         BEC;
END_REGION

REGION Network 3: Desconexión por finalización correcta
   // Si se mide un valor de velocidad fuera del rango, pero se corrige antes de que acabe el tiempo límite, se 
   // considera que la maniobra finaliza correctamente.
         A     #S7;
         S     #bdf_correcta;
   //R     #S7

         R     #bdt;
         R     #bde_velocidad;
         R     #Temporizador;
         FR    #Temporizador;
         R     #Sentido_antihorario;
         R     #fuera_rango;
         BEC;
END_REGION

REGION Network 4: Activación
         SET;
         FP    #bdt;

         R     #bdf_correcta;
         R     #bde_velocidad;

         S     #X1;
         R     #X2;
         R     #X_Err_Cinta;
         R     #S7;
END_REGION

REGION Network 5
         O     #X1;
         O     #X2;

         CALL  SCALE
         ( IN      := #vel_cinta_bits,
           HI_LIM  := 10000.0,
           LO_LIM  := 0.0,
           BIPOLAR := false,
           RET_VAL := #ret_val_scale,
           OUT     := #vel_cinta_rpm
         );
         O     #X1;
         O     #X2;
         A(;
         L     #ret_val_scale;
         L     W#16#0008;
         );
         ==I;
         =     #fuera_rango;
END_REGION

REGION Network 6: X1 ->X2
         A     #X1;
         A     #fuera_rango;
         S     #X2;
         R     #X1;
END_REGION

REGION Network 7: Configuración del temporizador
         A     #X2;
         L     #t_lim;
         SD    #Temporizador;
END_REGION

REGION Network 8: X2-> X_Err_Cinta
         A     #X2;
         A     #Temporizador;
         S     #X_Err_Cinta;
         R     #X2;
END_REGION

REGION Network 9: X2 -> S7
         A     #X2;
         AN    #fuera_rango;
         S     #S7;
         R     #X2;
END_REGION

REGION Network 10: Tratamiento de X1
         A     #X1;
         S     #Sentido_antihorario;
END_REGION

REGION Network 11: Tratamiento de X_Err_Cinta
         A     #X_Err_Cinta;
         R     #Sentido_antihorario;
END_REGION
END_FUNCTION_BLOCK

// folder: Emergencia

FUNCTION "Emergencia" : Void   // FC3, STL
{ S7_Optimized_Access := 'TRUE' }
VERSION : 0.1
BEGIN

REGION Network 1: Tratamiento de X_EMER
   // Se llama a todas las macroetapas, forzando como TRUE el valor de RESET, para que cada macroetapa haga la gestión de la emergencia.
         A     "EMER";
         JCN   _TratamientoEmergencia;
         CALL  "maniobra_barnizado", "maniobra_barnizado_DB"
         ( SP               := ,
           indicador_de_fin := ,
           t_lim            := ,
           Temporizador     := "Temp_barnizado",
           RESET            := true,
           Actuador         := "Barnizar",
           bde_tiempo       := "aviso_error_barnizado",
           bdf_correcta     := "aviso_fin_barnizado"
         );

         CALL  "maniobra_cinta", "maniobra_cinta_DB"
         ( vel_cinta_bits      := ,
           t_lim               := ,
           Temporizador        := "Temp_cinta",
           RESET               := true,
           Sentido_antihorario := "cinta_sentido_antihorario",
           bdf_correcta        := "aviso_fin_cinta",
           bde_velocidad       := "aviso_error_cinta"
         );

         CALL  "maniobra_grabado_secado", "maniobra_grabado_DB"
         ( SP_maq                   := ,
           t_normal_maq             := ,
           t_lim_man                := ,
           RESET                    := true,
           Temp_normal_maq          := "Temp_grabado_normal",
           Temp_lim_maq             := "Temp_grabado_lim",
           bdf_correcta             := "aviso_fin_grabado_p",
           bde_Tiempo               := "aviso_error_grabado_p",
           aviso_a_robot_para_coger := "aviso_al_pp_coger_pieza_grabado_p",
           Actuador                 := "Grabar"
         );

         CALL  "maniobra_grabado_secado", "maniobra_secado_DB"
         ( SP_maq                   := ,
           t_normal_maq             := ,
           t_lim_man                := ,
           RESET                    := true,
           Temp_normal_maq          := "Temp_secado1_normal",
           Temp_lim_maq             := "Temp_secado1_lim",
           bdf_correcta             := "aviso_fin_secado1",
           bde_Tiempo               := "aviso_error_secado1",
           aviso_a_robot_para_coger := "aviso_al_pp_coger_pieza_secado1",
           Actuador                 := "Secar"
         );

         CALL  "maniobra_pickandplace", "maniobra_pickandplace_DB"
         ( SP1          := ,
           P_cogida     := ,
           S_home       := ,
           t_lim        := ,
           Temporizador := "Temp_pickandplace",
           RESET        := true,
           SP2          := ,
           Mov1         := "Robot_coger",
           Mov2         := "Robot_delante",
           Mov4         := "Robot_reposo",
           bdf_correcta := "aviso_fin_pickandplace",
           bde_tiempo   := "aviso_errorT_pickandplace",
           bde_config   := "aviso_errorConf_pickandplace",
           Mov0         := "Robot_izq",
           Mov3         := "Robot_dejar"
         );


         CALL  "maniobra_pintado", "maniobra_pintado_DB_1"
         ( SP_pieza              := ,
           SP_lamina_mesa        := ,
           SP_lamina_pos_inicial := ,
           ModoLamina            := ,
           ModoNormal            := ,
           pintado_terminado     := ,
           RESET                 := true,
           t_lim_pintado_con_lam := ,
           t_lim_pintado_sin_lam := ,
           Temporizador_limite   := "Temp_pintado_lim",
           Tempor_pickandplace1  := "Temp_pickandplace",
           Tempor_pickandplace2  := "Temp_pickandplace",
           SP_pickandplace_in    := ,
           SP_pickandplace_out   := ,
           Sensor_home           := ,
           Lamina_cogida         := ,
           t_lim_pickandplace    := ,
           Act_pintar            := "Pintar",
           bde_tiempo            := "aviso_error_pintado",
           bdf_correcta          := "aviso_fin_pintado"
         );

         CALL  "maniobra_plataforma_omnidireccional", "maniobra_plataforma_omnidireccional_DB"
         ( SP                          := ,
           Lectura_correcta            := ,
           Lectura_incorrecta          := ,
           Entra_estacion              := ,
           Sigue_cinta                 := ,
           SP_estacion                 := ,
           RESET                       := true,
           t_lim_lectura               := ,
           t_lim_maniobra              := ,
           Temp_lectura                := "Temp_lectura_s1_in",
           Temp_maniobra               := "Temp_plataforma_s1",
           Actuador_ruedas_por_defecto := "giro_ruedas_por_defecto",
           Actuador_lectura            := "Leer",
           Actuador_ruedas_giro        := "giro_ruedas_izquierda",
           bde_tiempo_lectura          := "aviso_errorT_lectura_plataforma_s1",
           bde_tiempo                  := "aviso_errorT_lectura_plataforma_s1",
           bde_lectura                 := "aviso_error_lectura_plataforma",
           bdf_piezadentro             := "aviso_fin_entrada_s1",
           bdf_piezasiguerecto         := "aviso_fin_noEntra_s1"
         );

   _TratamientoEmergencia:NOP   0;

         A     "EMER";
         S     "X_EMER";

         R     "X1";
         R     "X2";
         R     "X3";
         R     "X4";
         R     "X5";
         R     "X6";
         R     "X_ON";
         R     "X_OFF";
         R     "X20";
         R     "X21";
         R     "X22";
         R     "X0";
         R     "XM1";
         R     "XM2";
         R     "XM3";
         R     "XM4";
         R     "XM5";
         R     "XM6";
         R     "X10";
         R     "X_PintadoModoCuadricula";
         R     "X_PintadoModoNormal";

         BEC;
END_REGION

REGION Network 2: Rearme de la celda mediante el pulsador de rearme sin estar la seta activada.
         A     "X_EMER";
         A     "rearme";
         AN    "EMER";
         S     "X0";
         R     "X_EMER";
END_REGION
END_FUNCTION

// folder: Entrada_a_estacion

FUNCTION_BLOCK "maniobra_plataforma_omnidireccional"   // FB7, STL
{ S7_Optimized_Access := 'TRUE' }
VERSION : 0.1
   VAR_INPUT
      SP : Bool;
      Lectura_correcta : Bool;
      Lectura_incorrecta : Bool;
      Entra_estacion : Bool;
      Sigue_cinta : Bool;
      SP_estacion : Bool;
      RESET : Bool;
      t_lim_lectura : S5Time;
      t_lim_maniobra : S5Time;
      Temp_lectura : Timer;
      Temp_maniobra : Timer;
   END_VAR
   VAR_OUTPUT
      Actuador_ruedas_por_defecto : Bool;
      Actuador_lectura : Bool;
      Actuador_ruedas_giro : Bool;
      bde_tiempo_lectura : Bool;
      bde_tiempo : Bool;
      bde_lectura : Bool;
      bdf_piezadentro : Bool;
      bdf_piezasiguerecto : Bool;
   END_VAR
   VAR
      XE5 : Bool;
      X1 : Bool;
      X2 : Bool;
      X3 : Bool;
      X4 : Bool;
      X_Err_TLectura : Bool;
      X_Err_Lectura : Bool;
      "XS5.1" : Bool;
      "XS5.2" : Bool;
      X_Err_Tiempo : Bool;
      bdt : Bool;
   END_VAR
BEGIN

REGION Network 1: Desconexión por RESET
         A     #RESET;

         R     #bdt;
         R     #bde_tiempo_lectura;
         R     #bdf_piezadentro;
         R     #bdf_piezasiguerecto;
         R     #bde_lectura;
         R     #bde_tiempo;

         R     #Temp_maniobra;
         FR    #Temp_maniobra;

         R     #Actuador_lectura;
         R     #Actuador_ruedas_giro;
         BEC;
END_REGION

REGION Network 2: Desconexión por error síncrono
         A     #X_Err_Tiempo;
         S     #bde_tiempo;
   //R     #X_Err_Tiempo

         R     #bdt;
         R     #bde_tiempo_lectura;
         R     #bdf_piezadentro;
         R     #bdf_piezasiguerecto;
         R     #bde_lectura;

         R     #Temp_maniobra;
         FR    #Temp_maniobra;

         R     #Actuador_lectura;
         R     #Actuador_ruedas_giro;
         BEC;
END_REGION

REGION Network 3: Desconexión por error por mala lectura
         A     #X_Err_Lectura;
         S     #bde_lectura;
   // R     #X_Err_Lectura

         R     #bdt;
         R     #bde_tiempo_lectura;
         R     #bdf_piezadentro;
         R     #bdf_piezasiguerecto;
         R     #bde_tiempo;

         R     #Temp_maniobra;
         FR    #Temp_maniobra;

         R     #Actuador_lectura;
         R     #Actuador_ruedas_giro;
         BEC;
END_REGION

REGION Network 4: Desconexión por error síncrono de lectura
         A     #X_Err_TLectura;
         S     #bde_tiempo_lectura;
   // R     #X_Err_TLectura

         R     #bdt;
         R     #bde_lectura;
         R     #bdf_piezadentro;
         R     #bdf_piezasiguerecto;
         R     #bde_tiempo;

         R     #Temp_maniobra;
         FR    #Temp_maniobra;

         R     #Actuador_lectura;
         R     #Actuador_ruedas_giro;
         BEC;
END_REGION

REGION Network 5: Desconexión por finalización correcta (pieza entra a la estación)
         A     #"XS5.1";
         S     #bdf_piezadentro;
   // R     #"XS5.1"

         R     #bdt;
         R     #bde_tiempo_lectura;
         R     #bdf_piezasiguerecto;
         R     #bde_lectura;
         R     #bde_tiempo;

         R     #Temp_maniobra;
         FR    #Temp_maniobra;

         R     #Actuador_lectura;
         R     #Actuador_ruedas_giro;
         BEC;
END_REGION

REGION Network 6: Desconexión por finalización correcta (pieza NO entra a la estación y sigue recto)
         A     #"XS5.2";
         S     #bdf_piezasiguerecto;
   //R     #"XS5.2"

         R     #bdt;
         R     #bde_tiempo_lectura;
         R     #bdf_piezadentro;
         R     #bde_lectura;
         R     #bde_tiempo;

         R     #Temp_maniobra;
         FR    #Temp_maniobra;

         R     #Actuador_lectura;
         R     #Actuador_ruedas_giro;
         BEC;
END_REGION

REGION Network 7: Conexión
         SET;
         FP    #bdt;

         R     #bdf_piezadentro;
         R     #bde_lectura;
         R     #bde_tiempo_lectura;
         R     #bde_tiempo;
         R     #bdf_piezasiguerecto;

         S     #XE5;
         S     #Actuador_ruedas_por_defecto;
         R     #X1;
         R     #X2;
         R     #X3;
         R     #"XS5.1";
         R     #"XS5.2";
         R     #X_Err_Lectura;
         R     #X_Err_Tiempo;
END_REGION

REGION Network 8: E5 -> X1
         A     #XE5;
         A     #SP;
         S     #X1;
         R     #XE5;
END_REGION

REGION Network 9: Configuración del perro guardián
         A     #X1;

         L     #t_lim_maniobra;
         SS    #Temp_maniobra;

         L     #t_lim_lectura;
         SD    #Temp_lectura;
END_REGION

REGION Network 10: X1 -> X_Err_Lectura
         A     #X1;
         A     #Temp_lectura;
         S     #X_Err_TLectura;
         R     #X1;
END_REGION

REGION Network 11: X1 -> X2
         A     #X1;
         A     #Lectura_correcta;
         AN    #Temp_lectura;
         S     #X2;
         R     #X1;
END_REGION

REGION Network 12: X1->X4
         A     #X1;
         A     #Lectura_incorrecta;
         AN    #Temp_lectura;
         S     #X4;
         R     #X1;
END_REGION

REGION Network 13: X2 -> X3
         A     #X2;
         A     #Entra_estacion;
         S     #X3;
         R     #X2;
         R     #Actuador_ruedas_por_defecto;
END_REGION

REGION Network 14: X3 -> S5.1
         A     #X3;
         A     #SP_estacion;
         R     #X3;
         S     #Actuador_ruedas_por_defecto;
         S     #"XS5.1";
END_REGION

REGION Network 15: X2 -> S5.2
         A     #X2;
         A     #Sigue_cinta;
         S     #"XS5.2";
         R     #X2;
END_REGION

REGION Network 16: Activación del perro guardián
         A     #Temp_maniobra;
         =     #X_Err_Tiempo;
END_REGION

REGION Network 17: Tratamiento X1
         A     #X1;
         =     #Actuador_lectura;
END_REGION

REGION Network 18: Tratamiento X3
         A     #X3;
         =     #Actuador_ruedas_giro;
END_REGION

REGION Network 19: Tratamiento X4
         A     #X4;
         =     #X_Err_Lectura;
END_REGION
END_FUNCTION_BLOCK

// folder: Flancos

FUNCTION "Flancos" : Void   // FC2, STL
{ S7_Optimized_Access := 'TRUE' }
VERSION : 0.1
BEGIN

REGION Network 1
         A     "ON";
         FP    "M_flanco";
         =     "PON";
END_REGION
END_FUNCTION

// folder: Grabado_y_secado

FUNCTION_BLOCK "maniobra_grabado_secado"   // FB3, STL
{ S7_Optimized_Access := 'TRUE' }
VERSION : 0.1
   VAR_INPUT
      SP_maq : Bool;
      t_normal_maq : S5Time;
      t_lim_man : S5Time;
      RESET : Bool;
      Temp_normal_maq : Timer;
      Temp_lim_maq : Timer;
   END_VAR
   VAR_OUTPUT
      bdf_correcta : Bool;
      bde_Tiempo : Bool;
      aviso_a_robot_para_coger : Bool;
      Actuador : Bool;
   END_VAR
   VAR
      XE3 : Bool;
      X1 : Bool;
      X2 : Bool;
      XS3 : Bool;
      X_Err_Tiempo_Man : Bool;
      bdt : Bool;
   END_VAR
BEGIN

REGION Network 1: Desconexión por RESET
         A     #RESET;

         R     #bdt;
         R     #bde_Tiempo;
         R     #bdf_correcta;

         R     #Temp_lim_maq;
         R     #Temp_normal_maq;
         FR    #Temp_lim_maq;
         FR    #Temp_normal_maq;

         R     #Actuador;
         R     #aviso_a_robot_para_coger;
         BEC;
END_REGION

REGION Network 2: Desonexión por error síncrono (exceso de tiempo en la maniobra de grabado o secado)
         A     #X_Err_Tiempo_Man;
         S     #bde_Tiempo;
   // R     #X_Err_Tiempo_Man

         R     #bdt;
         R     #bdf_correcta;

         R     #Temp_lim_maq;
         R     #Temp_normal_maq;
         FR    #Temp_lim_maq;
         FR    #Temp_normal_maq;

         R     #Actuador;
         R     #aviso_a_robot_para_coger;
         BEC;
END_REGION

REGION Network 3: Desconexión por finalización correcta de maniobra
         A     #XS3;
         S     #bdf_correcta;
   //R     #XS3
         R     #bdt;
         R     #bde_Tiempo;

         R     #Temp_lim_maq;
         R     #Temp_normal_maq;
         FR    #Temp_lim_maq;
         FR    #Temp_normal_maq;

         R     #Actuador;
         R     #aviso_a_robot_para_coger;
         BEC;
END_REGION

REGION Network 4: Conexión
         SET;
         FP    #bdt;

         R     #bde_Tiempo;
         R     #bdf_correcta;

         S     #XE3;
         R     #X1;
         R     #X2;
         R     #XS3;
         R     #X_Err_Tiempo_Man;
END_REGION

REGION Network 5: E3 -> X1
         A     #XE3;
         A     #SP_maq;
         S     #X1;
         R     #XE3;
END_REGION

REGION Network 6
         A     #X1;
         L     #t_normal_maq;
         SD    #Temp_normal_maq;

         L     #t_lim_man;
         SS    #Temp_lim_maq;
END_REGION

REGION Network 7: X1 -> X2
         A     #X1;
         A     #Temp_normal_maq;
         S     #X2;
         R     #X1;
END_REGION

REGION Network 8: X2 -> S3
         A     #X2;
         AN    #SP_maq;
         S     #XS3;
         R     #X2;
END_REGION

REGION Network 9: Activación del perro guardián por exceso de tiempo
         A     #Temp_lim_maq;
         =     #X_Err_Tiempo_Man;
END_REGION

REGION Network 10: Tratamiento de X1
         A     #X1;
         =     #Actuador;
END_REGION

REGION Network 11: Tratamiento de X2
         A     #X2;
         =     #aviso_a_robot_para_coger;
END_REGION
END_FUNCTION_BLOCK

// folder: Pick_and_place

FUNCTION_BLOCK "maniobra_pickandplace"   // FB4, STL
{ S7_Optimized_Access := 'TRUE' }
VERSION : 0.1
   VAR_INPUT
      SP1 : Bool;
      P_cogida : Bool;
      S_home : Bool;
      t_lim : S5Time;
      Temporizador : Timer;
      RESET : Bool;
      SP2 : Bool;
   END_VAR
   VAR_OUTPUT
      Mov1 : Bool;
      Mov2 : Bool;
      Mov4 : Bool;
      bdf_correcta : Bool;
      bde_tiempo : Bool;
      bde_config : Bool;
      Mov0 : Bool;
      Mov3 : Bool;
   END_VAR
   VAR
      XE4 : Bool;
      X1 : Bool;
      X2 : Bool;
      X3 : Bool;
      X4 : Bool;
      XS4 : Bool;
      X_Err_Tiempo : Bool;
      X_Err_Config : Bool;
      bdt : Bool;
   END_VAR
BEGIN

REGION Network 1: Desconexión por RESET
         A     #RESET;
   //resetar los bits
         R     #bdt;
         R     #bde_tiempo;
         R     #bde_config;
         R     #bdf_correcta;
   //resetar temporizador
         R     #Temporizador;
         FR    #Temporizador;
   //resetar actuadores
         R     #Mov0;
         R     #Mov1;
         R     #Mov2;
         R     #Mov3;
         R     #Mov4;
         BEC;
END_REGION

REGION Network 2: Desconexión por error síncrono
         A     #X_Err_Tiempo;
         S     #bde_tiempo;
   //R     #X_Err_Tiempo
         R     #bdt;
         R     #bdf_correcta;
         R     #bde_config;
         R     #Temporizador;
         FR    #Temporizador;
         R     #Mov0;
         R     #Mov1;
         R     #Mov2;
         R     #Mov3;
         R     #Mov4;
         BEC;
END_REGION

REGION Network 3: Desconexión por error de configuración
         A     #X_Err_Config;
         S     #bde_config;
   // R     #X_Err_Config
         R     #bdt;
         R     #bde_tiempo;
         R     #bdf_correcta;
         R     #Temporizador;
         FR    #Temporizador;
         R     #Mov0;
         R     #Mov1;
         R     #Mov2;
         R     #Mov3;
         R     #Mov4;

         BEC;
END_REGION

REGION Network 4: Desconexión por finalización correcta
         A     #XS4;
         S     #bdf_correcta;
   //R     #XS4
         R     #bdt;
         R     #bde_tiempo;
         R     #bde_config;
         R     #Temporizador;
         FR    #Temporizador;
         R     #Mov0;
         R     #Mov1;
         R     #Mov2;
         R     #Mov3;
         R     #Mov4;
         BEC;
END_REGION

REGION Network 5: Conexión
         SET;
         FP    #bdt;
         R     #bdf_correcta;
         R     #bde_config;
         R     #bde_tiempo;

         S     #XE4;
         R     #X1;
         R     #X2;
         R     #X3;
         R     #X4;
         R     #XS4;
         R     #X_Err_Config;
         R     #X_Err_Tiempo;
END_REGION

REGION Network 6: E4 -> X1
         A     #XE4;
         A     #SP1;
         S     #X1;
         R     #XE4;
END_REGION

REGION Network 7: Configuración del perro guardián
         A     #X4;  //cambiar a otro estado al finalizar test Q SINO NO ME DABA TIEMPO
         L     #t_lim;
         SS    #Temporizador;
END_REGION

REGION Network 8: X1 -> X2
         A     #X1;
         A     #P_cogida;
         S     #X2;
         R     #X1;
END_REGION

REGION Network 9: X2 -> X_Err_Config
   // Error por mala configuración: se produce cuando no se detecta la pieza cogida, cuando previamente se detectaba y no ha sido depositada,
   // es decir, cuando se cae de las pinzas.
         A     #X2;
         AN    #P_cogida;
         S     #X_Err_Config;
         R     #X2;
END_REGION

REGION Network 10: X2 -> X3
         A     #X2;
         A     #SP2;
         S     #X3;
         R     #X2;
END_REGION

REGION Network 11: X3 -> X4
         A     #X3;
         AN    #P_cogida;
         S     #X4;
         R     #X3;
END_REGION

REGION Network 12: X4 -> S4
         A     #X4;
         A     #S_home;
         S     #XS4;
         R     #X4;
END_REGION

REGION Network 13: Activación de perro guardián
         A     #Temporizador;
         =     #X_Err_Tiempo;
END_REGION

REGION Network 14
         A     #XE4;
         =     #Mov0;
END_REGION

REGION Network 15: Tratamiento de X1
         A     #X1;
         =     #Mov1;
END_REGION

REGION Network 16: Tratamiento de X2
         A     #X2;
         =     #Mov2;
END_REGION

REGION Network 17: Tratamiento de X3
         A     #X3;
         =     #Mov3;
END_REGION

REGION Network 18: Tratamiento de X4
         A     #X4;
         =     #Mov4;
END_REGION
END_FUNCTION_BLOCK

// folder: Pintado

FUNCTION_BLOCK "maniobra_pintado"   // FB6, STL
{ S7_Optimized_Access := 'TRUE' }
VERSION : 0.1
   VAR_INPUT
      SP_pieza : Bool;
      SP_lamina_mesa : Bool;
      SP_lamina_pos_inicial : Bool;
      ModoLamina : Bool;
      ModoNormal : Bool;
      pintado_terminado : Bool;
      RESET : Bool;
      t_lim_pintado_con_lam : S5Time;
      t_lim_pintado_sin_lam : S5Time;
      Temporizador_limite : Timer;
      Tempor_pickandplace1 : Timer;
      Tempor_pickandplace2 : Timer;
      SP_pickandplace_in : Bool;
      SP_pickandplace_out : Bool;
      Sensor_home : Bool;
      Lamina_cogida : Bool;
      t_lim_pickandplace : S5Time;
   END_VAR
   VAR_OUTPUT
      Act_pintar : Bool;
      bde_tiempo : Bool;
      bdf_correcta : Bool;
   END_VAR
   VAR
      usar_lamina : "maniobra_pickandplace";
      guardar_lamina : "maniobra_pickandplace";
      XE1 : Bool;
      X1 : Bool;
      XM1 : Bool;
      XM2 : Bool;
      X2 : Bool;
      X3 : Bool;
      XS1 : Bool;
      X_Err_Tiempo : Bool;
      bdt : Bool;
      Robot_lam_izq : Bool;
      Robot_lam_coger : Bool;
      Robot_lam_delante : Bool;
      Robot_lam_dejar : Bool;
      Robot_lam_dcha : Bool;
      Robot_lam_reposo : Bool;
   END_VAR
   VAR_TEMP
      fin_usar_lamina : Bool;
      fin_guardar_lamina : Bool;
      errorT_usar_lamina : Bool;
      errorConf_usar_lamina : Bool;
      errorT_guardar_lamina : Bool;
      errorConf_guardar_lamina : Bool;
   END_VAR
BEGIN

REGION Network 1: Desconexión por RESET
   // Resetea la FB de pintado, y llama a la FB de instancia de pick and place.
         A     #RESET;
         R     #bdt;
         R     #bde_tiempo;
         R     #bdf_correcta;

         R     #Temporizador_limite;
         FR    #Temporizador_limite;
         R     #Act_pintar;
         JCN   _ResetPickAndPlace;
         CALL  #usar_lamina
         ( SP1          := ,
           P_cogida     := ,
           S_home       := ,
           t_lim        := ,
           Temporizador := ,
           RESET        := true,
           SP2          := ,
           Mov1         := #Robot_lam_coger,
           Mov2         := #Robot_lam_delante,
           Mov4         := #Robot_lam_reposo,
           bdf_correcta := #fin_usar_lamina,
           bde_tiempo   := #errorT_usar_lamina,
           bde_config   := #errorConf_usar_lamina,
           Mov0         := #Robot_lam_izq,
           Mov3         := #Robot_lam_dejar
         );

         CALL  #guardar_lamina
         ( SP1          := ,
           P_cogida     := ,
           S_home       := ,
           t_lim        := ,
           Temporizador := ,
           RESET        := true,
           SP2          := ,
           Mov1         := #Robot_lam_coger,
           Mov2         := #Robot_lam_dcha,
           Mov4         := #Robot_lam_reposo,
           bdf_correcta := #fin_guardar_lamina,
           bde_tiempo   := #errorT_guardar_lamina,
           bde_config   := #errorConf_guardar_lamina,
           Mov0         := #Robot_lam_delante,
           Mov3         := #Robot_lam_dejar
         );


   _ResetPickAndPlace:NOP   0;

         A     #RESET;
         BEC;
END_REGION

REGION Network 2: Desconexión por error síncrono
         A     #X_Err_Tiempo;
         S     #bde_tiempo;
         R     #X_Err_Tiempo;

         R     #bdt;
         R     #bdf_correcta;
         R     #Temporizador_limite;
         FR    #Temporizador_limite;

         R     #Act_pintar;
         BEC;
END_REGION

REGION Network 3
         A     #XS1;
         S     #bdf_correcta;
         R     #XS1;

         R     #bdt;
         R     #bde_tiempo;
         R     #Temporizador_limite;
         FR    #Temporizador_limite;

         R     #Act_pintar;
         BEC;
END_REGION

REGION Network 4: Conexión/Arranque de la FB
         SET;
         FP    #bdt;
         R     #bdf_correcta;
         R     #bde_tiempo;
         S     #XE1;
         R     #X1;
         R     #XM1;
         R     #X2;
         R     #XM2;
         R     #X3;
         R     #XS1;
         R     #X_Err_Tiempo;
END_REGION

REGION Network 5: E1 -> X1
         A     #XE1;
         A     #SP_pieza;
         S     #X1;
         R     #XE1;
END_REGION

REGION Network 6: X1 -> X3
   // Pintado normal, es decir, únicamente consta de un robot de pintado que pulveriza spray sobre la pieza.
         A     #X1;
         A     #ModoNormal;
         S     #X3;
         R     #X1;
END_REGION

REGION Network 7: Perro guardián para el modo de pintado normal (sin lámina)
         A     #X3;
         JCN   _tiempo_lim_pintado_sin_lamina;
         L     #t_lim_pintado_sin_lam;
         SS    #Temporizador_limite;

   _tiempo_lim_pintado_sin_lamina:NOP   0;
END_REGION

REGION Network 8: X3 -> S1
         A     #X3;
         A     #pintado_terminado;
         S     #XS1;
         R     #X3;
END_REGION

REGION Network 9: X1 -> M1 (maniobra de dejar la lámina sobre la pieza)
         A     #X1;
         A     #ModoLamina;
         S     #XM1;
         R     #X1;
END_REGION

REGION Network 10: Perro guardián para el modo de pintado con lámina (tablero de ajedrez)
         A     #XM1;
         JCN   _tiempo_lim_pintado_con_lamina;
         L     #t_lim_pintado_con_lam;
         SS    #Temporizador_limite;
   _tiempo_lim_pintado_con_lamina:NOP   0;
END_REGION

REGION Network 11: X2 -> XM2
         A     #X2;
         A     #pintado_terminado;
         S     #XM2;
         R     #X2;
END_REGION

REGION Network 12: Tratamiento M1 y M1 -> X2
         A     #XM1;
         JCN   _maniobra_usar_lamina;
         CALL  #usar_lamina
         ( SP1          := #SP_lamina_pos_inicial,
           P_cogida     := #Lamina_cogida,
           S_home       := #Sensor_home,
           t_lim        := #t_lim_pickandplace,
           Temporizador := #Tempor_pickandplace1,
           RESET        := false,
           SP2          := #SP_lamina_mesa,
           Mov1         := #Robot_lam_coger,
           Mov2         := #Robot_lam_delante,
           Mov4         := #Robot_lam_reposo,
           bdf_correcta := #fin_usar_lamina,
           bde_tiempo   := #errorT_usar_lamina,
           bde_config   := #errorConf_usar_lamina,
           Mov0         := #Robot_lam_izq,
           Mov3         := #Robot_lam_dejar
         );

         A     #errorT_usar_lamina;
         S     #X_Err_Tiempo;
         R     #XM1;

         A     #fin_usar_lamina;
         S     #X2;
         R     #XM1;
   _maniobra_usar_lamina:NOP   0;
END_REGION

REGION Network 13: Tratamiento de M2 y M2 -> S1
         A     #XM2;
         JCN   _maniobra_guardar_lamina;
         CALL  #guardar_lamina
         ( SP1          := #SP_lamina_mesa,
           P_cogida     := #Lamina_cogida,
           S_home       := #Sensor_home,
           t_lim        := #t_lim_pickandplace,
           Temporizador := #Tempor_pickandplace2,
           RESET        := false,
           SP2          := #SP_lamina_pos_inicial,
           Mov1         := #Robot_lam_coger,
           Mov2         := #Robot_lam_dcha,
           Mov4         := #Robot_lam_reposo,
           bdf_correcta := #fin_guardar_lamina,
           bde_tiempo   := #errorT_guardar_lamina,
           bde_config   := #errorConf_guardar_lamina,
           Mov0         := #Robot_lam_delante,
           Mov3         := #Robot_lam_dejar
         );
         A     #errorT_guardar_lamina;
         S     #X_Err_Tiempo;
         R     #XM2;

         A     #fin_guardar_lamina;
         S     #XS1;
         R     #XM2;

   _maniobra_guardar_lamina:NOP   0;
END_REGION

REGION Network 14: Activación de perro guardián por exceso de tiempo en las maniobras de pick and place o en la propia maniobra de pintado
         A     #Temporizador_limite;
         O     #Tempor_pickandplace1;
         O     #Tempor_pickandplace2;
         S     #X_Err_Tiempo;
END_REGION

REGION Network 15: Tratamiento de X2 y X3
         O     #X2;
         O     #X3;
         =     #Act_pintar;
END_REGION
END_FUNCTION_BLOCK

FUNCTION_BLOCK "Pintado"   // FB6, STL
{ S7_Optimized_Access := 'TRUE' }
VERSION : 0.1
   VAR_INPUT
      SP_pieza : Bool;
      SP_lamina_mesa : Bool;
      SP_lamina_pos_inicial : Bool;
      ModoLamina : Bool;
      ModoNormal : Bool;
      pintado_terminado : Bool;
      t_lim_pintado_con_lam : S5Time;
      EMER : Bool;
      rearme : Bool;
      START : Bool;
      t_lim_pintado_sin_lam : S5Time;
      Temp_lim_pintado : Timer;
      Tempor_pickandplace_usar : Timer;
      Tempor_pickandplace_guardar : Timer;
      SP_pickandplace_in : Bool;
      SP_pickandplace_out : Bool;
      Sensor_home : Bool;
      Lamina_cogida : Bool;
      t_lim_pickandplace : S5Time;
   END_VAR
   VAR_OUTPUT
      Act_pintar : Bool;
      bde_tiempo : Bool;
      bit_stdby : Bool;
      bit_emer : Bool;
      bde_pickandplace : Bool;
   END_VAR
   VAR
      usar_lamina : "maniobra_pickandplace";
      guardar_lamina : "maniobra_pickandplace";
      X_Init : Bool;
      X_Stdby : Bool;
      XM1 : Bool;
      XM2 : Bool;
      X3 : Bool;
      X4 : Bool;
      X2 : Bool;
      X_Err_Tiempo : Bool;
      X_Err_PickAndPlace : Bool;
      X_Emer : Bool;
      bit_trabajo : Bool;
      Robot_lam_izq : Bool;
      Robot_lam_coger : Bool;
      Robot_lam_delante : Bool;
      Robot_lam_dejar : Bool;
      Robot_lam_dcha : Bool;
      Robot_lam_reposo : Bool;
   END_VAR
   VAR_TEMP
      fin_usar_lamina : Bool;
      fin_guardar_lamina : Bool;
      errorT_usar_lamina : Bool;
      errorConf_usar_lamina : Bool;
      errorT_guardar_lamina : Bool;
      errorConf_guardar_lamina : Bool;
   END_VAR
BEGIN

REGION Network 1: Desconexión por RESET
   // Resetea la FB de pintado, y llama a la FB de instancia de pick and place.
         AN    #START;
         R     #bit_trabajo;
         R     #bde_tiempo;
         R     #bit_stdby;
         R     #bit_emer;
         R     #bde_pickandplace;

         R     #Temp_lim_pintado;
         FR    #Temp_lim_pintado;
         R     #Act_pintar;
         JCN   _ResetPickAndPlace;
         CALL  #usar_lamina
         ( SP1          := ,
           P_cogida     := ,
           S_home       := ,
           t_lim        := ,
           Temporizador := ,
           RESET        := true,
           SP2          := ,
           Mov1         := #Robot_lam_coger,
           Mov2         := #Robot_lam_delante,
           Mov4         := #Robot_lam_reposo,
           bdf_correcta := #fin_usar_lamina,
           bde_tiempo   := #errorT_usar_lamina,
           bde_config   := #errorConf_usar_lamina,
           Mov0         := #Robot_lam_izq,
           Mov3         := #Robot_lam_dejar
         );

         CALL  #guardar_lamina
         ( SP1          := ,
           P_cogida     := ,
           S_home       := ,
           t_lim        := ,
           Temporizador := ,
           RESET        := true,
           SP2          := ,
           Mov1         := #Robot_lam_coger,
           Mov2         := #Robot_lam_dcha,
           Mov4         := #Robot_lam_reposo,
           bdf_correcta := #fin_guardar_lamina,
           bde_tiempo   := #errorT_guardar_lamina,
           bde_config   := #errorConf_guardar_lamina,
           Mov0         := #Robot_lam_delante,
           Mov3         := #Robot_lam_dejar
         );


   _ResetPickAndPlace:NOP   0;

         AN    #START;
         BEC;
END_REGION

REGION Network 2: Conexión/Arranque de la FB
         SET;
         FP    #bit_trabajo;

         R     #bde_tiempo;
         R     #bit_emer;
         R     #bde_pickandplace;


         S     #X_Stdby;
         R     #X_Init;
         R     #X2;
         R     #XM1;
         R     #X3;
         R     #XM2;
         R     #X4;
         R     #X_Err_Tiempo;
         R     #X_Emer;
         R     #X_Err_PickAndPlace;
END_REGION

REGION Network 3: X_Stdby -> X2
         A     #X_Stdby;
         A     #SP_pieza;
         S     #X2;
         R     #X_Stdby;
END_REGION

REGION Network 4: X2 -> X4
   // Pintado normal, es decir, únicamente consta de un robot de pintado que pulveriza spray sobre la pieza.
         A     #X2;
         A     #ModoNormal;
         S     #X4;
         R     #X2;
END_REGION

REGION Network 5: Perro guardián para el modo de pintado normal (sin lámina)
         A     #X4;
         JCN   _tiempo_lim_pintado_sin_lamina;
         L     #t_lim_pintado_sin_lam;
         SS    #Temp_lim_pintado;

   _tiempo_lim_pintado_sin_lamina:NOP   0;
END_REGION

REGION Network 6: X3 -> S1
         A     #X4;
         A     #pintado_terminado;
         S     #X_Stdby;
         R     #X4;
END_REGION

REGION Network 7: X2 -> M1 (maniobra de dejar la lámina sobre la pieza)
         A     #X2;
         A     #ModoLamina;
         S     #XM1;
         R     #X2;
END_REGION

REGION Network 8: Perro guardián para el modo de pintado con lámina (tablero de ajedrez)
         A     #XM1;
         JCN   _tiempo_lim_pintado_con_lamina;
         L     #t_lim_pintado_con_lam;
         SS    #Temp_lim_pintado;
   _tiempo_lim_pintado_con_lamina:NOP   0;
END_REGION

REGION Network 9: X3 -> XM2
         A     #X3;
         A     #pintado_terminado;
         S     #XM2;
         R     #X3;
END_REGION

REGION Network 10: Tratamiento M1 y M1 -> X3
         A     #XM1;
         JCN   _maniobra_usar_lamina;
         CALL  #usar_lamina
         ( SP1          := #SP_lamina_pos_inicial,
           P_cogida     := #Lamina_cogida,
           S_home       := #Sensor_home,
           t_lim        := #t_lim_pickandplace,
           Temporizador := #Tempor_pickandplace_usar,
           RESET        := false,
           SP2          := #SP_lamina_mesa,
           Mov1         := #Robot_lam_coger,
           Mov2         := #Robot_lam_delante,
           Mov4         := #Robot_lam_reposo,
           bdf_correcta := #fin_usar_lamina,
           bde_tiempo   := #errorT_usar_lamina,
           bde_config   := #errorConf_usar_lamina,
           Mov0         := #Robot_lam_izq,
           Mov3         := #Robot_lam_dejar
         );

         A     #errorT_usar_lamina;
         O     #errorConf_usar_lamina;
         S     #X_Err_PickAndPlace;
         R     #XM1;

         A     #fin_usar_lamina;
         S     #X3;
         R     #XM1;
   _maniobra_usar_lamina:NOP   0;
END_REGION

REGION Network 11: Tratamiento de M2 y M2 -> X1 ("X_stdby")
         A     #XM2;
         JCN   _maniobra_guardar_lamina;
         CALL  #guardar_lamina
         ( SP1          := #SP_lamina_mesa,
           P_cogida     := #Lamina_cogida,
           S_home       := #Sensor_home,
           t_lim        := #t_lim_pickandplace,
           Temporizador := #Tempor_pickandplace_guardar,
           RESET        := false,
           SP2          := #SP_lamina_pos_inicial,
           Mov1         := #Robot_lam_coger,
           Mov2         := #Robot_lam_dcha,
           Mov4         := #Robot_lam_reposo,
           bdf_correcta := #fin_guardar_lamina,
           bde_tiempo   := #errorT_guardar_lamina,
           bde_config   := #errorConf_guardar_lamina,
           Mov0         := #Robot_lam_delante,
           Mov3         := #Robot_lam_dejar
         );

         A     #errorT_guardar_lamina;
         O     #errorConf_guardar_lamina;
         S     #X_Err_PickAndPlace;
         R     #XM2;

         A     #fin_guardar_lamina;
         S     #X_Stdby;
         R     #XM2;

   _maniobra_guardar_lamina:NOP   0;
END_REGION

REGION Network 12: Activación de perro guardián por exceso de tiempo en la unidad productiva de pintado
         A     #Temp_lim_pintado;
         S     #X_Err_Tiempo;
END_REGION

REGION Network 13: Tratamiento de X3 y X4
         O     #X3;
         O     #X4;
         =     #Act_pintar;
END_REGION

REGION Network 14: Desconexión por error síncrono (error de tiempo de la unidad productiva)
         A     #X_Err_Tiempo;
         =     #bde_tiempo;

         JCN   _informar_maniobras_error_sincrono;
         CALL  #usar_lamina
         ( SP1          := ,
           P_cogida     := ,
           S_home       := ,
           t_lim        := ,
           Temporizador := #Tempor_pickandplace_usar,
           RESET        := true,
           SP2          := ,
           Mov1         := #Robot_lam_coger,
           Mov2         := #Robot_lam_delante,
           Mov4         := #Robot_lam_reposo,
           bdf_correcta := #fin_usar_lamina,
           bde_tiempo   := #errorT_usar_lamina,
           bde_config   := #errorConf_usar_lamina,
           Mov0         := #Robot_lam_izq,
           Mov3         := #Robot_lam_dejar
         );

         CALL  #guardar_lamina
         ( SP1          := ,
           P_cogida     := ,
           S_home       := ,
           t_lim        := ,
           Temporizador := #Tempor_pickandplace_guardar,
           RESET        := true,
           SP2          := ,
           Mov1         := #Robot_lam_coger,
           Mov2         := #Robot_lam_dcha,
           Mov4         := #Robot_lam_reposo,
           bdf_correcta := #fin_guardar_lamina,
           bde_tiempo   := #errorT_guardar_lamina,
           bde_config   := #errorConf_guardar_lamina,
           Mov0         := #Robot_lam_delante,
           Mov3         := #Robot_lam_dejar
         );

   _informar_maniobras_error_sincrono:NOP   0;
END_REGION

REGION Network 15: Desconexión por error síncrono (errores de las maniobras pick and place)
         A     #X_Err_PickAndPlace;
         =     #bde_pickandplace;

         JCN   _informar_maniobras_error_sincrono_pickandplace;
         CALL  #usar_lamina
         ( SP1          := ,
           P_cogida     := ,
           S_home       := ,
           t_lim        := ,
           Temporizador := #Tempor_pickandplace_usar,
           RESET        := true,
           SP2          := ,
           Mov1         := #Robot_lam_coger,
           Mov2         := #Robot_lam_delante,
           Mov4         := #Robot_lam_reposo,
           bdf_correcta := #fin_usar_lamina,
           bde_tiempo   := #errorT_usar_lamina,
           bde_config   := #errorConf_usar_lamina,
           Mov0         := #Robot_lam_izq,
           Mov3         := #Robot_lam_dejar
         );

         CALL  #guardar_lamina
         ( SP1          := ,
           P_cogida     := ,
           S_home       := ,
           t_lim        := ,
           Temporizador := #Tempor_pickandplace_guardar,
           RESET        := true,
           SP2          := ,
           Mov1         := #Robot_lam_coger,
           Mov2         := #Robot_lam_dcha,
           Mov4         := #Robot_lam_reposo,
           bdf_correcta := #fin_guardar_lamina,
           bde_tiempo   := #errorT_guardar_lamina,
           bde_config   := #errorConf_guardar_lamina,
           Mov0         := #Robot_lam_delante,
           Mov3         := #Robot_lam_dejar
         );

   _informar_maniobras_error_sincrono_pickandplace:NOP   0;
END_REGION

REGION Network 16: Rearme de los estados de error
         A(;
         O     #X_Err_Tiempo;
         O     #X_Err_PickAndPlace;
         );
         A     #rearme;
         R     #X_Err_Tiempo;
         R     #X_Err_PickAndPlace;
         S     #X_Stdby;
END_REGION

REGION Network 17: Activación de X_Emer
         A     #EMER;
         S     #X_Emer;

         R     #X_Init;
         R     #X_Stdby;
         R     #X2;
         R     #X3;
         R     #X4;
         R     #XM1;
         R     #XM2;
END_REGION

REGION Network 18: Tratamiento de X_Emer
         A     #X_Emer;
         =     #bit_emer;

         JCN   _informar_maniobras_de_emer;
         CALL  #usar_lamina
         ( SP1          := ,
           P_cogida     := ,
           S_home       := ,
           t_lim        := ,
           Temporizador := #Tempor_pickandplace_usar,
           RESET        := true,
           SP2          := ,
           Mov1         := #Robot_lam_coger,
           Mov2         := #Robot_lam_delante,
           Mov4         := #Robot_lam_reposo,
           bdf_correcta := #fin_usar_lamina,
           bde_tiempo   := #errorT_usar_lamina,
           bde_config   := #errorConf_usar_lamina,
           Mov0         := #Robot_lam_izq,
           Mov3         := #Robot_lam_dejar
         );

         CALL  #guardar_lamina
         ( SP1          := ,
           P_cogida     := ,
           S_home       := ,
           t_lim        := ,
           Temporizador := #Tempor_pickandplace_guardar,
           RESET        := true,
           SP2          := ,
           Mov1         := #Robot_lam_coger,
           Mov2         := #Robot_lam_dcha,
           Mov4         := #Robot_lam_reposo,
           bdf_correcta := #fin_guardar_lamina,
           bde_tiempo   := #errorT_guardar_lamina,
           bde_config   := #errorConf_guardar_lamina,
           Mov0         := #Robot_lam_delante,
           Mov3         := #Robot_lam_dejar
         );

   _informar_maniobras_de_emer:NOP   0;
END_REGION

REGION Network 19: Rearme desde X_Emer (X_Emer -> X1)
         A     #X_Emer;
         A     #rearme;
         AN    #EMER;
         S     #X_Stdby;
         R     #X_Emer;
END_REGION

REGION Network 20: Activación del bit de standby
         A     #X_Stdby;
         =     #bit_stdby;
END_REGION
END_FUNCTION_BLOCK

// folder: Produccion

FUNCTION "Modos_pintado" : Void   // FC1, STL
TITLE = Grafcet de modos de pintado
{ S7_Optimized_Access := 'TRUE' }
VERSION : 0.1
// Si se activa el sensor de presencia y sensor de lectura detecta un tablero de ajedrez, se activa el pintado modo cuadrícula, que se define en el FB de pintado. Si no, se activa el pintado modo normal.
BEGIN

REGION Network 1: X10 -> X_PintadoModoCuadricula
         A     "X10";
         A     "SP_pintado_PiezaEnMesa";
         A     "Tablero_ajedrez";
         S     "X_PintadoModoCuadricula";
         R     "X10";
END_REGION

REGION Network 2: X_PintadoModoCuadricula -> X10
         A     "X_PintadoModoCuadricula";
         A     "aviso_fin_pintado";
         S     "X10";
         R     "X_PintadoModoCuadricula";
END_REGION

REGION Network 3: X10 -> X_PintadoModoNormal
         A     "X10";
         A     "SP_pintado_PiezaEnMesa";
         AN    "Tablero_ajedrez";
         S     "X_PintadoModoNormal";
         R     "X10";
END_REGION

REGION Network 4: X_PintadoModoNormal -> X10
         A     "X_PintadoModoNormal";
         A     "aviso_fin_pintado";
         S     "X10";
         R     "X_PintadoModoNormal";
END_REGION

REGION Network 5: Tratamiento de X_PintadoModoCuadricula
         A     "X_PintadoModoCuadricula";
         JCN   _001;
         L     "Datos_ModoCuadricula".t_lim_pintado_ModoCuadricula;
         T     "Datos_produccion".t_lim_pintado;
   _001: NOP   0;
END_REGION

REGION Network 6: Tratamiento de X_PintadoModoNormal
         A     "X_PintadoModoNormal";
         JCN   _002;
         L     "Datos_ModoNormal".t_lim_pintado_ModoNormal;
         T     "Datos_produccion".t_lim_pintado;
   _002: NOP   0;
END_REGION
END_FUNCTION

FUNCTION "contador_fallos_lectura" : Void   // FC11, STL
{ S7_Optimized_Access := 'TRUE' }
VERSION : 0.1
   VAR_INPUT
      max_malas_lecturas : Word;
   END_VAR
   VAR_OUTPUT
      debe_retirar_piezas : Bool;
   END_VAR
BEGIN

REGION Network 1
         A     "X20";
         L     C#0;
         S     "Contador_lecturas_defectuosas";
END_REGION

REGION Network 2
         A(;
         L     "Contador_lecturas_defectuosas";  // carga en el ACU2
         L     #max_malas_lecturas;  // CARGA EN ACU 1
         ==I;  //RLO a 1 si ACU1=ACU2 COMPARANDO ENTEROS
         );
         =     #debe_retirar_piezas;
END_REGION

REGION Network 3
         A     "X21";
         CU    "Contador_lecturas_defectuosas";
END_REGION
END_FUNCTION

FUNCTION "gestion_fallos_lectura" : Void   // FC12, STL
{ S7_Optimized_Access := 'TRUE' }
VERSION : 0.1
BEGIN

REGION Network 1: X20->X21
         A     "X20";
         A     "lectura_defectuosa";
         R     "X20";
         S     "X21";
END_REGION

REGION Network 2: ACTIVACIÓN TEMPORIZADOR EN X21
         A     "X21";
         L     "Datos_produccion".t_fugaz_21;
         SD    "Temp_fugaz_21";
END_REGION

REGION Network 3: X21->X22
         A     "X21";
         A     "Temp_fugaz_21";
         S     "X22";
         R     "X21";
END_REGION

REGION Network 4: X22->X21
         A     "X22";
         A     "lectura_defectuosa";
         AN    "evento_lecturas";
         S     "X21";
         R     "X22";
END_REGION

REGION Network 5: X22->X23
         A     "X22";
         A     "evento_lecturas";
         R     "X22";
         S     "X23";
END_REGION

REGION Network 6: X23->X20
         A     "X23";
         A     "rearme";
         S     "X20";
         R     "X23";
END_REGION

REGION Network 7
         A     "X23";
         =     "Luz_Roja";
END_REGION
END_FUNCTION

// folder: Tests_unitarios

FUNCTION "test_barnizado" : Void   // FC4, STL
{ S7_Optimized_Access := 'TRUE' }
VERSION : 0.1
BEGIN

REGION Network 1
         CALL  "maniobra_barnizado", "maniobra_barnizado_DB"
         ( SP               := "SP_barnizado_in",
           indicador_de_fin := "SP_barnizado_out",
           t_lim            := "Datos_produccion".t_lim_barnizado,
           Temporizador     := "Temp_barnizado",
           RESET            := false,
           Actuador         := "Barnizar",
           bde_tiempo       := "aviso_error_barnizado",
           bdf_correcta     := "aviso_fin_barnizado"
         );
END_REGION
END_FUNCTION

FUNCTION "test_secado" : Void   // FC5, STL
{ S7_Optimized_Access := 'TRUE' }
VERSION : 0.1
BEGIN

REGION Network 1
         CALL  "maniobra_grabado_secado", "maniobra_secado_DB"
         ( SP_maq                   := "SP_secado1",
           t_normal_maq             := "Datos_produccion".t_normal_secado,
           t_lim_man                := "Datos_produccion".t_lim_secado,
           RESET                    := false,
           Temp_normal_maq          := "Temp_secado1_normal",
           Temp_lim_maq             := "Temp_secado1_lim",
           bdf_correcta             := "aviso_fin_secado1",
           bde_Tiempo               := "aviso_error_secado1",
           aviso_a_robot_para_coger := "aviso_al_pp_coger_pieza_secado1",
           Actuador                 := "Secar"
         );
END_REGION
END_FUNCTION

FUNCTION "test_pickandplace" : Void   // FC6, STL
{ S7_Optimized_Access := 'TRUE' }
VERSION : 0.1
BEGIN

REGION Network 1: Test unitario del robot pick and place de la celda de secado 1
   // Test para el movimiento de robot al entrar una pieza en la estación de secado.
   // El movimiento es el siguiente: al robot le entra una pieza por la izquierda ("robot_izq"), la coge, la deja en la máquina ("robot_delante") y vuelve
   // su estado de reposo.
         CALL  "maniobra_pickandplace", "maniobra_pickandplace_DB"
         ( SP1          := "SP_pickandplace_s1_in",
           P_cogida     := "Pieza_cogida_robpp_s1",
           S_home       := "Home_robpp_s1",
           t_lim        := "Datos_produccion".t_lim_pickandplace,
           Temporizador := "Temp_pickandplace_s1",
           RESET        := FALSE,
           SP2          := "SP_secado1",
           Mov1         := "Robot_coger",
           Mov2         := "Robot_delante",
           Mov4         := "Robot_reposo",
           bdf_correcta := "aviso_fin_pickandplace",
           bde_tiempo   := "aviso_errorT_pickandplace",
           bde_config   := "aviso_errorConf_pickandplace",
           Mov0         := "Robot_izq",
           Mov3         := "Robot_dejar"
         );
END_REGION
END_FUNCTION

FUNCTION "test_grabado" : Void   // FC7, STL
{ S7_Optimized_Access := 'TRUE' }
VERSION : 0.1
BEGIN

REGION Network 1
         CALL  "maniobra_grabado_secado", "maniobra_grabado_DB"
         ( SP_maq                   := "SP_grabado_p",
           t_normal_maq             := "Datos_produccion".t_normal_grabado,
           t_lim_man                := "Datos_produccion".t_lim_grabado,
           RESET                    := FALSE,
           Temp_normal_maq          := "Temp_grabado_normal",
           Temp_lim_maq             := "Temp_grabado_lim",
           bdf_correcta             := "aviso_fin_grabado_p",
           bde_Tiempo               := "aviso_error_grabado_p",
           aviso_a_robot_para_coger := "aviso_al_pp_coger_pieza_grabado_p",
           Actuador                 := "Grabar"
         );
END_REGION
END_FUNCTION

FUNCTION "test_plataforma_omnidireccional" : Void   // FC8, STL
{ S7_Optimized_Access := 'TRUE' }
VERSION : 0.1
BEGIN

REGION Network 1
         CALL  "maniobra_plataforma_omnidireccional", "maniobra_plataforma_omnidireccional_DB"
         ( SP                          := "SP_lectura_s1",
           Lectura_correcta            := "lectura_correcta_s1",
           Lectura_incorrecta          := "lectura_incorrecta_s1",
           Entra_estacion              := "entra_s1",
           Sigue_cinta                 := "sigue_s1",
           SP_estacion                 := "SP_secado1",
           RESET                       := false,
           t_lim_lectura               := "Datos_produccion".t_lim_respuesta_lectura,
           t_lim_maniobra              := "Datos_produccion".t_lim_plat_omni,
           Temp_lectura                := "Temp_plataforma_lectura_s1",
           Temp_maniobra               := "Temp_plataforma_s1",
           Actuador_ruedas_por_defecto := "giro_ruedas_por_defecto",
           Actuador_lectura            := "Leer",
           Actuador_ruedas_giro        := "giro_ruedas_izquierda",
           bde_tiempo_lectura          := "aviso_errorT_lectura_plataforma_s1",
           bde_tiempo                  := "avisor_errorT_plataforma_s1",
           bde_lectura                 := "aviso_error_lectura_plataforma",
           bdf_piezadentro             := "aviso_fin_entrada_s1",
           bdf_piezasiguerecto         := "aviso_fin_noEntra_s1"
         );
END_REGION
END_FUNCTION

FUNCTION "test_pintado" : Void   // FC9, STL
{ S7_Optimized_Access := 'TRUE' }
VERSION : 0.1
BEGIN

REGION Network 1

         CALL  "maniobra_pintado", "maniobra_pintado_DB_1"
         ( SP_pieza              := "SP_pintado_PiezaEnMesa",
           SP_lamina_mesa        := "SP_pintado_LaminaEnMesa",
           SP_lamina_pos_inicial := "SP_pintado_LaminaEnOrigen",
           ModoLamina            := "X_PintadoModoCuadricula",
           ModoNormal            := "X_PintadoModoNormal",
           pintado_terminado     := "fin_pintado",
           RESET                 := false,
           t_lim_pintado_con_lam := "Datos_produccion".t_lim_pintado_ModoCuadricula,
           t_lim_pintado_sin_lam := "Datos_produccion".t_lim_pintado_ModoNormal,
           Temporizador_limite   := "Temp_pintado_lim",
           Tempor_pickandplace1  := "Temp_pickandplace",
           Tempor_pickandplace2  := "Temp_pickandplace",
           SP_pickandplace_in    := "SP_pickandplace_p_in",
           SP_pickandplace_out   := "SP_pickandplace_p_out",
           Sensor_home           := "Home_robpp_p",
           Lamina_cogida         := "Pieza_cogida",
           t_lim_pickandplace    := "Datos_produccion".t_lim_pickandplace,
           Act_pintar            := "Pintar",
           bde_tiempo            := "aviso_error_pintado",
           bdf_correcta          := "aviso_fin_pintado"
         );
END_REGION
END_FUNCTION

FUNCTION "test_cinta" : Void   // FC10, STL
{ S7_Optimized_Access := 'TRUE' }
VERSION : 0.1
BEGIN

REGION Network 1
         CALL  "maniobra_cinta", "maniobra_cinta_DB"
         ( vel_cinta_bits      := "vel_cinta_muestreada_bits",
           t_lim               := "Datos_produccion".t_lim_cinta,
           Temporizador        := "Temp_cinta",
           RESET               := "EMER",
           Sentido_antihorario := "cinta_sentido_antihorario",
           bdf_correcta        := "aviso_fin_cinta",
           bde_velocidad       := "aviso_error_cinta"
         );
END_REGION
END_FUNCTION